  STRUCT
   FAC1_IF : STRUCT
    FAC_COMM_CHECK : INT ;	//FAC-PLC통신 확인용 정보 FAC=11,PLC=1
    PLC_ONLINE_MODE : INT ;	//생산지시 ON_OFF선택 정보 ON=1,OFF=0
    STATION_WORK_COMPLETE : INT ;	//공정 작업완료 정보 ON=1,OFF=0
    PLC_DATA_REQ_COUNT : INT ;	//차종 요청 카운터
    FINAL_SEND_VINDATA1 : WORD ;	//공정 최종 사용 VIN1
    FINAL_SEND_VINDATA2 : WORD ;	//공정 최종 사용 VIN2
    RCV_DATA_CHECK_ERROR : INT ;	//수신 데이터 CHECK이상 이상=1,정상=0
    RESERVED1 : INT ;
    RESERVED2 : INT ;
    RESERVED3 : INT ;
    LINE_DATA_READ_REQ : INT ;	//라인 현황 반영 요청 PLC=1,FAC=11
    ORDER_DATA_REQ : INT ;	//차종 설정 요청 PLC=1,FAC=11(정상처리),11<> 이상처리,99=서열부족,100=강제설정
    PRESENT_VIN_DATA1 : WORD ;	//차종 설정 데이터(현재)
    PRESENT_VIN_DATA2 : WORD ;	//차종 설정 데이터(현재)
    PRESENT_BODY_DATA1 : WORD ;	//차종 설정 데이터(현재)
    PRESENT_BODY_DATA2 : WORD ;	//차종 설정 데이터(현재)
    PRESENT_BODY_DATA3 : WORD ;	//차종 설정 데이터(현재)
    PRESENT_BODY_DATA4 : WORD ;	//차종 설정 데이터(현재)
    PRESENT_RESERVED_DATA1 : WORD ;	//차종 설정 데이터(현재)
    PRESENT_RESERVED_DATA2 : WORD ;	//차종 설정 데이터(현재)
    NEXT_VIN_DATA1 : WORD ;	//차종 설정 데이터(다음)
    NEXT_VIN_DATA2 : WORD ;	//차종 설정 데이터(다음)
    NEXT_BODY_DATA1 : WORD ;	//차종 설정 데이터(다음)
    NEXT_BODY_DATA2 : WORD ;	//차종 설정 데이터(다음)
    NEXT_BODY_DATA3 : WORD ;	//차종 설정 데이터(다음)
    NEXT_BODY_DATA4 : WORD ;	//차종 설정 데이터(다음)
    NEXT_RESERVED_DATA1 : WORD ;	//차종 설정 데이터(다음)
    NEXT_RESERVED_DATA2 : WORD ;	//차종 설정 데이터(다음)
    RESERVED4 : WORD ;
    RESERVED5 : WORD ;
   END_STRUCT ;
   FAC2_IF : STRUCT
    FAC_COMM_CHECK : INT ;	//FAC-PLC통신 확인용 정보 FAC=11,PLC=1
    PLC_ONLINE_MODE : INT ;	//생산지시 ON_OFF선택 정보 ON=1,OFF=0
    STATION_WORK_COMPLETE : INT ;	//공정 작업완료 정보 ON=1,OFF=0
    PLC_DATA_REQ_COUNT : INT ;	//차종 요청 카운터
    FINAL_SEND_VINDATA1 : WORD ;	//공정 최종 사용 VIN1
    FINAL_SEND_VINDATA2 : WORD ;	//공정 최종 사용 VIN2
    RCV_DATA_CHECK_ERROR : INT ;	//수신 데이터 CHECK이상 이상=1,정상=0
    RESERVED1 : INT ;
    RESERVED2 : INT ;
    CMP_ORDER_DATA_REQ : INT ;	//차종 설정 요청 정보 변경 내용 확인용
    LINE_DATA_READ_REQ : INT ;	//라인 현황 반영 요청 PLC=1,FAC=11
    ORDER_DATA_REQ : INT ;	//차종 설정 요청 PLC=1,FAC=11(정상처리),11<> 이상처리,99=서열부족,100=강제설정
    PRESENT_VIN_DATA1 : WORD ;	//차종 설정 데이터(현재)
    PRESENT_VIN_DATA2 : WORD ;	//차종 설정 데이터(현재)
    PRESENT_BODY_DATA1 : WORD ;	//차종 설정 데이터(현재)
    PRESENT_BODY_DATA : WORD ;	//차종 설정 데이터(현재)
    PRESENT_BODY_DATA3 : WORD ;	//차종 설정 데이터(현재)
    PRESENT_BODY_DATA4 : WORD ;	//차종 설정 데이터(현재)
    PRESENT_RESERVED_DATA1 : WORD ;	//차종 설정 데이터(현재)
    PRESENT_RESERVED_DATA2 : WORD ;	//차종 설정 데이터(현재)
    NEXT_VIN_DATA1 : WORD ;	//차종 설정 데이터(다음)
    NEXT_VIN_DATA2 : WORD ;	//차종 설정 데이터(다음)
    NEXT_BODY_DATA1 : WORD ;	//차종 설정 데이터(다음)
    NEXT_BODY_DATA2 : WORD ;	//차종 설정 데이터(다음)
    NEXT_BODY_DATA3 : WORD ;	//차종 설정 데이터(다음)
    NEXT_BODY_DATA4 : WORD ;	//차종 설정 데이터(다음)
    NEXT_RESERVED_DATA1 : WORD ;	//차종 설정 데이터(다음)
    NEXT_RESERVED_DATA2 : WORD ;	//차종 설정 데이터(다음)
    RESERVED4 : WORD ;
    RESERVED5 : WORD ;
   END_STRUCT ;
   FAC3_IF : STRUCT
    FAC_COMM_CHECK : INT ;	//FAC-PLC통신 확인용 정보 FAC=11,PLC=1
    PLC_ONLINE_MODE : INT ;	//생산지시 ON_OFF선택 정보 ON=1,OFF=0
    STATION_WORK_COMPLETE : INT ;	//공정 작업완료 정보 ON=1,OFF=0
    PLC_DATA_REQ_COUNT : INT ;	//차종 요청 카운터
    FINAL_SEND_VINDATA1 : WORD ;	//공정 최종 사용 VIN1
    FINAL_SEND_VINDATA2 : WORD ;	//공정 최종 사용 VIN2
    RCV_DATA_CHECK_ERROR : INT ;	//수신 데이터 CHECK이상 이상=1,정상=0
    RESERVED1 : INT ;
    RESERVED2 : INT ;
    CMP_ORDER_DATA_REQ : INT ;	//차종 설정 요청 정보 변경 내용 확인용
    LINE_DATA_READ_REQ : INT ;	//라인 현황 반영 요청 PLC=1,FAC=11
    ORDER_DATA_REQ : INT ;	//차종 설정 요청 PLC=1,FAC=11(정상처리),11<> 이상처리,99=서열부족,100=강제설정
    PRESENT_VIN_DATA1 : WORD ;	//차종 설정 데이터(현재)
    PRESENT_VIN_DATA2 : WORD ;	//차종 설정 데이터(현재)
    PRESENT_BODY_DATA1 : WORD ;	//차종 설정 데이터(현재)
    PRESENT_BODY_DATA : WORD ;	//차종 설정 데이터(현재)
    PRESENT_BODY_DATA3 : WORD ;	//차종 설정 데이터(현재)
    PRESENT_BODY_DATA4 : WORD ;	//차종 설정 데이터(현재)
    PRESENT_RESERVED_DATA1 : WORD ;	//차종 설정 데이터(현재)
    PRESENT_RESERVED_DATA2 : WORD ;	//차종 설정 데이터(현재)
    NEXT_VIN_DATA1 : WORD ;	//차종 설정 데이터(다음)
    NEXT_VIN_DATA2 : WORD ;	//차종 설정 데이터(다음)
    NEXT_BODY_DATA1 : WORD ;	//차종 설정 데이터(다음)
    NEXT_BODY_DATA2 : WORD ;	//차종 설정 데이터(다음)
    NEXT_BODY_DATA3 : WORD ;	//차종 설정 데이터(다음)
    NEXT_BODY_DATA4 : WORD ;	//차종 설정 데이터(다음)
    NEXT_RESERVED_DATA1 : WORD ;	//차종 설정 데이터(다음)
    NEXT_RESERVED_DATA2 : WORD ;	//차종 설정 데이터(다음)
    RESERVED4 : WORD ;
    RESERVED5 : WORD ;
   END_STRUCT ;
   FAC4_IF : STRUCT
    FAC_COMM_CHECK : INT ;	//FAC-PLC통신 확인용 정보 FAC=11,PLC=1
    PLC_ONLINE_MODE : INT ;	//생산지시 ON_OFF선택 정보 ON=1,OFF=0
    STATION_WORK_COMPLETE : INT ;	//공정 작업완료 정보 ON=1,OFF=0
    PLC_DATA_REQ_COUNT : INT ;	//차종 요청 카운터
    FINAL_SEND_VINDATA1 : WORD ;	//공정 최종 사용 VIN1
    FINAL_SEND_VINDATA2 : WORD ;	//공정 최종 사용 VIN2
    RCV_DATA_CHECK_ERROR : INT ;	//수신 데이터 CHECK이상 이상=1,정상=0
    RESERVED1 : INT ;
    RESERVED2 : INT ;
    CMP_ORDER_DATA_REQ : INT ;	//차종 설정 요청 정보 변경 내용 확인용
    LINE_DATA_READ_REQ : INT ;	//라인 현황 반영 요청 PLC=1,FAC=11
    ORDER_DATA_REQ : INT ;	//차종 설정 요청 PLC=1,FAC=11(정상처리),11<> 이상처리,99=서열부족,100=강제설정
    PRESENT_VIN_DATA1 : WORD ;	//차종 설정 데이터(현재)
    PRESENT_VIN_DATA2 : WORD ;	//차종 설정 데이터(현재)
    PRESENT_BODY_DATA1 : WORD ;	//차종 설정 데이터(현재)
    PRESENT_BODY_DATA : WORD ;	//차종 설정 데이터(현재)
    PRESENT_BODY_DATA3 : WORD ;	//차종 설정 데이터(현재)
    PRESENT_BODY_DATA4 : WORD ;	//차종 설정 데이터(현재)
    PRESENT_RESERVED_DATA1 : WORD ;	//차종 설정 데이터(현재)
    PRESENT_RESERVED_DATA2 : WORD ;	//차종 설정 데이터(현재)
    NEXT_VIN_DATA1 : WORD ;	//차종 설정 데이터(다음)
    NEXT_VIN_DATA2 : WORD ;	//차종 설정 데이터(다음)
    NEXT_BODY_DATA1 : WORD ;	//차종 설정 데이터(다음)
    NEXT_BODY_DATA2 : WORD ;	//차종 설정 데이터(다음)
    NEXT_BODY_DATA3 : WORD ;	//차종 설정 데이터(다음)
    NEXT_BODY_DATA4 : WORD ;	//차종 설정 데이터(다음)
    NEXT_RESERVED_DATA1 : WORD ;	//차종 설정 데이터(다음)
    NEXT_RESERVED_DATA2 : WORD ;	//차종 설정 데이터(다음)
    RESERVED4 : WORD ;
    RESERVED5 : WORD ;
   END_STRUCT ;
   FAC5_IF : STRUCT
    FAC_COMM_CHECK : INT ;	//FAC-PLC통신 확인용 정보 FAC=11,PLC=1
    PLC_ONLINE_MODE : INT ;	//생산지시 ON_OFF선택 정보 ON=1,OFF=0
    STATION_WORK_COMPLETE : INT ;	//공정 작업완료 정보 ON=1,OFF=0
    PLC_DATA_REQ_COUNT : INT ;	//차종 요청 카운터
    FINAL_SEND_VINDATA1 : WORD ;	//공정 최종 사용 VIN1
    FINAL_SEND_VINDATA2 : WORD ;	//공정 최종 사용 VIN2
    RCV_DATA_CHECK_ERROR : INT ;	//수신 데이터 CHECK이상 이상=1,정상=0
    RESERVED1 : INT ;
    RESERVED2 : INT ;
    CMP_ORDER_DATA_REQ : INT ;	//차종 설정 요청 정보 변경 내용 확인용
    LINE_DATA_READ_REQ : INT ;	//라인 현황 반영 요청 PLC=1,FAC=11
    ORDER_DATA_REQ : INT ;	//차종 설정 요청 PLC=1,FAC=11(정상처리),11<> 이상처리,99=서열부족,100=강제설정
    PRESENT_VIN_DATA1 : WORD ;	//차종 설정 데이터(현재)
    PRESENT_VIN_DATA2 : WORD ;	//차종 설정 데이터(현재)
    PRESENT_BODY_DATA1 : WORD ;	//차종 설정 데이터(현재)
    PRESENT_BODY_DATA : WORD ;	//차종 설정 데이터(현재)
    PRESENT_BODY_DATA3 : WORD ;	//차종 설정 데이터(현재)
    PRESENT_BODY_DATA4 : WORD ;	//차종 설정 데이터(현재)
    PRESENT_RESERVED_DATA1 : WORD ;	//차종 설정 데이터(현재)
    PRESENT_RESERVED_DATA2 : WORD ;	//차종 설정 데이터(현재)
    NEXT_VIN_DATA1 : WORD ;	//차종 설정 데이터(다음)
    NEXT_VIN_DATA2 : WORD ;	//차종 설정 데이터(다음)
    NEXT_BODY_DATA1 : WORD ;	//차종 설정 데이터(다음)
    NEXT_BODY_DATA2 : WORD ;	//차종 설정 데이터(다음)
    NEXT_BODY_DATA3 : WORD ;	//차종 설정 데이터(다음)
    NEXT_BODY_DATA4 : WORD ;	//차종 설정 데이터(다음)
    NEXT_RESERVED_DATA1 : WORD ;	//차종 설정 데이터(다음)
    NEXT_RESERVED_DATA2 : WORD ;	//차종 설정 데이터(다음)
    RESERVED4 : WORD ;
    RESERVED5 : WORD ;
   END_STRUCT ;
   FAC6_IF : STRUCT
    FAC_COMM_CHECK : INT ;	//FAC-PLC통신 확인용 정보 FAC=11,PLC=1
    PLC_ONLINE_MODE : INT ;	//생산지시 ON_OFF선택 정보 ON=1,OFF=0
    STATION_WORK_COMPLETE : INT ;	//공정 작업완료 정보 ON=1,OFF=0
    PLC_DATA_REQ_COUNT : INT ;	//차종 요청 카운터
    FINAL_SEND_VINDATA1 : WORD ;	//공정 최종 사용 VIN1
    FINAL_SEND_VINDATA2 : WORD ;	//공정 최종 사용 VIN2
    RCV_DATA_CHECK_ERROR : INT ;	//수신 데이터 CHECK이상 이상=1,정상=0
    RESERVED1 : INT ;
    RESERVED2 : INT ;
    CMP_ORDER_DATA_REQ : INT ;	//차종 설정 요청 정보 변경 내용 확인용
    LINE_DATA_READ_REQ : INT ;	//라인 현황 반영 요청 PLC=1,FAC=11
    ORDER_DATA_REQ : INT ;	//차종 설정 요청 PLC=1,FAC=11(정상처리),11<> 이상처리,99=서열부족,100=강제설정
    PRESENT_VIN_DATA1 : WORD ;	//차종 설정 데이터(현재)
    PRESENT_VIN_DATA2 : WORD ;	//차종 설정 데이터(현재)
    PRESENT_BODY_DATA1 : WORD ;	//차종 설정 데이터(현재)
    PRESENT_BODY_DATA : WORD ;	//차종 설정 데이터(현재)
    PRESENT_BODY_DATA3 : WORD ;	//차종 설정 데이터(현재)
    PRESENT_BODY_DATA4 : WORD ;	//차종 설정 데이터(현재)
    PRESENT_RESERVED_DATA1 : WORD ;	//차종 설정 데이터(현재)
    PRESENT_RESERVED_DATA2 : WORD ;	//차종 설정 데이터(현재)
    NEXT_VIN_DATA1 : WORD ;	//차종 설정 데이터(다음)
    NEXT_VIN_DATA2 : WORD ;	//차종 설정 데이터(다음)
    NEXT_BODY_DATA1 : WORD ;	//차종 설정 데이터(다음)
    NEXT_BODY_DATA2 : WORD ;	//차종 설정 데이터(다음)
    NEXT_BODY_DATA3 : WORD ;	//차종 설정 데이터(다음)
    NEXT_BODY_DATA4 : WORD ;	//차종 설정 데이터(다음)
    NEXT_RESERVED_DATA1 : WORD ;	//차종 설정 데이터(다음)
    NEXT_RESERVED_DATA2 : WORD ;	//차종 설정 데이터(다음)
    RESERVED4 : WORD ;
    RESERVED5 : WORD ;
   END_STRUCT ;
   FAC7_IF : STRUCT
    FAC_COMM_CHECK : INT ;	//FAC-PLC통신 확인용 정보 FAC=11,PLC=1
    PLC_ONLINE_MODE : INT ;	//생산지시 ON_OFF선택 정보 ON=1,OFF=0
    STATION_WORK_COMPLETE : INT ;	//공정 작업완료 정보 ON=1,OFF=0
    PLC_DATA_REQ_COUNT : INT ;	//차종 요청 카운터
    FINAL_SEND_VINDATA1 : WORD ;	//공정 최종 사용 VIN1
    FINAL_SEND_VINDATA2 : WORD ;	//공정 최종 사용 VIN2
    RCV_DATA_CHECK_ERROR : INT ;	//수신 데이터 CHECK이상 이상=1,정상=0
    RESERVED1 : INT ;
    RESERVED2 : INT ;
    CMP_ORDER_DATA_REQ : INT ;	//차종 설정 요청 정보 변경 내용 확인용
    LINE_DATA_READ_REQ : INT ;	//라인 현황 반영 요청 PLC=1,FAC=11
    ORDER_DATA_REQ : INT ;	//차종 설정 요청 PLC=1,FAC=11(정상처리),11<> 이상처리,99=서열부족,100=강제설정
    PRESENT_VIN_DATA1 : WORD ;	//차종 설정 데이터(현재)
    PRESENT_VIN_DATA2 : WORD ;	//차종 설정 데이터(현재)
    PRESENT_BODY_DATA1 : WORD ;	//차종 설정 데이터(현재)
    PRESENT_BODY_DATA : WORD ;	//차종 설정 데이터(현재)
    PRESENT_BODY_DATA3 : WORD ;	//차종 설정 데이터(현재)
    PRESENT_BODY_DATA4 : WORD ;	//차종 설정 데이터(현재)
    PRESENT_RESERVED_DATA1 : WORD ;	//차종 설정 데이터(현재)
    PRESENT_RESERVED_DATA2 : WORD ;	//차종 설정 데이터(현재)
    NEXT_VIN_DATA1 : WORD ;	//차종 설정 데이터(다음)
    NEXT_VIN_DATA2 : WORD ;	//차종 설정 데이터(다음)
    NEXT_BODY_DATA1 : WORD ;	//차종 설정 데이터(다음)
    NEXT_BODY_DATA2 : WORD ;	//차종 설정 데이터(다음)
    NEXT_BODY_DATA3 : WORD ;	//차종 설정 데이터(다음)
    NEXT_BODY_DATA4 : WORD ;	//차종 설정 데이터(다음)
    NEXT_RESERVED_DATA1 : WORD ;	//차종 설정 데이터(다음)
    NEXT_RESERVED_DATA2 : WORD ;	//차종 설정 데이터(다음)
    RESERVED4 : WORD ;
    RESERVED5 : WORD ;
   END_STRUCT ;
   FAC8_IF : STRUCT
    FAC_COMM_CHECK : INT ;	//FAC-PLC통신 확인용 정보 FAC=11,PLC=1
    PLC_ONLINE_MODE : INT ;	//생산지시 ON_OFF선택 정보 ON=1,OFF=0
    STATION_WORK_COMPLETE : INT ;	//공정 작업완료 정보 ON=1,OFF=0
    PLC_DATA_REQ_COUNT : INT ;	//차종 요청 카운터
    FINAL_SEND_VINDATA1 : WORD ;	//공정 최종 사용 VIN1
    FINAL_SEND_VINDATA2 : WORD ;	//공정 최종 사용 VIN2
    RCV_DATA_CHECK_ERROR : INT ;	//수신 데이터 CHECK이상 이상=1,정상=0
    RESERVED1 : INT ;
    RESERVED2 : INT ;
    CMP_ORDER_DATA_REQ : INT ;	//차종 설정 요청 정보 변경 내용 확인용
    LINE_DATA_READ_REQ : INT ;	//라인 현황 반영 요청 PLC=1,FAC=11
    ORDER_DATA_REQ : INT ;	//차종 설정 요청 PLC=1,FAC=11(정상처리),11<> 이상처리,99=서열부족,100=강제설정
    PRESENT_VIN_DATA1 : WORD ;	//차종 설정 데이터(현재)
    PRESENT_VIN_DATA2 : WORD ;	//차종 설정 데이터(현재)
    PRESENT_BODY_DATA1 : WORD ;	//차종 설정 데이터(현재)
    PRESENT_BODY_DATA : WORD ;	//차종 설정 데이터(현재)
    PRESENT_BODY_DATA3 : WORD ;	//차종 설정 데이터(현재)
    PRESENT_BODY_DATA4 : WORD ;	//차종 설정 데이터(현재)
    PRESENT_RESERVED_DATA1 : WORD ;	//차종 설정 데이터(현재)
    PRESENT_RESERVED_DATA2 : WORD ;	//차종 설정 데이터(현재)
    NEXT_VIN_DATA1 : WORD ;	//차종 설정 데이터(다음)
    NEXT_VIN_DATA2 : WORD ;	//차종 설정 데이터(다음)
    NEXT_BODY_DATA1 : WORD ;	//차종 설정 데이터(다음)
    NEXT_BODY_DATA2 : WORD ;	//차종 설정 데이터(다음)
    NEXT_BODY_DATA3 : WORD ;	//차종 설정 데이터(다음)
    NEXT_BODY_DATA4 : WORD ;	//차종 설정 데이터(다음)
    NEXT_RESERVED_DATA1 : WORD ;	//차종 설정 데이터(다음)
    NEXT_RESERVED_DATA2 : WORD ;	//차종 설정 데이터(다음)
    RESERVED4 : WORD ;
    RESERVED5 : WORD ;
   END_STRUCT ;
   FAC9_IF : STRUCT
    FAC_COMM_CHECK : INT ;	//FAC-PLC통신 확인용 정보 FAC=11,PLC=1
    PLC_ONLINE_MODE : INT ;	//생산지시 ON_OFF선택 정보 ON=1,OFF=0
    STATION_WORK_COMPLETE : INT ;	//공정 작업완료 정보 ON=1,OFF=0
    PLC_DATA_REQ_COUNT : INT ;	//차종 요청 카운터
    FINAL_SEND_VINDATA1 : WORD ;	//공정 최종 사용 VIN1
    FINAL_SEND_VINDATA2 : WORD ;	//공정 최종 사용 VIN2
    RCV_DATA_CHECK_ERROR : INT ;	//수신 데이터 CHECK이상 이상=1,정상=0
    RESERVED1 : INT ;
    RESERVED2 : INT ;
    CMP_ORDER_DATA_REQ : INT ;	//차종 설정 요청 정보 변경 내용 확인용
    LINE_DATA_READ_REQ : INT ;	//라인 현황 반영 요청 PLC=1,FAC=11
    ORDER_DATA_REQ : INT ;	//차종 설정 요청 PLC=1,FAC=11(정상처리),11<> 이상처리,99=서열부족,100=강제설정
    PRESENT_VIN_DATA1 : WORD ;	//차종 설정 데이터(현재)
    PRESENT_VIN_DATA2 : WORD ;	//차종 설정 데이터(현재)
    PRESENT_BODY_DATA1 : WORD ;	//차종 설정 데이터(현재)
    PRESENT_BODY_DATA : WORD ;	//차종 설정 데이터(현재)
    PRESENT_BODY_DATA3 : WORD ;	//차종 설정 데이터(현재)
    PRESENT_BODY_DATA4 : WORD ;	//차종 설정 데이터(현재)
    PRESENT_RESERVED_DATA1 : WORD ;	//차종 설정 데이터(현재)
    PRESENT_RESERVED_DATA2 : WORD ;	//차종 설정 데이터(현재)
    NEXT_VIN_DATA1 : WORD ;	//차종 설정 데이터(다음)
    NEXT_VIN_DATA2 : WORD ;	//차종 설정 데이터(다음)
    NEXT_BODY_DATA1 : WORD ;	//차종 설정 데이터(다음)
    NEXT_BODY_DATA2 : WORD ;	//차종 설정 데이터(다음)
    NEXT_BODY_DATA3 : WORD ;	//차종 설정 데이터(다음)
    NEXT_BODY_DATA4 : WORD ;	//차종 설정 데이터(다음)
    NEXT_RESERVED_DATA1 : WORD ;	//차종 설정 데이터(다음)
    NEXT_RESERVED_DATA2 : WORD ;	//차종 설정 데이터(다음)
    RESERVED4 : WORD ;
    RESERVED5 : WORD ;
   END_STRUCT ;
   FAC10_IF : STRUCT
    FAC_COMM_CHECK : INT ;	//FAC-PLC통신 확인용 정보 FAC=11,PLC=1
    PLC_ONLINE_MODE : INT ;	//생산지시 ON_OFF선택 정보 ON=1,OFF=0
    STATION_WORK_COMPLETE : INT ;	//공정 작업완료 정보 ON=1,OFF=0
    PLC_DATA_REQ_COUNT : INT ;	//차종 요청 카운터
    FINAL_SEND_VINDATA1 : WORD ;	//공정 최종 사용 VIN1
    FINAL_SEND_VINDATA2 : WORD ;	//공정 최종 사용 VIN2
    RCV_DATA_CHECK_ERROR : INT ;	//수신 데이터 CHECK이상 이상=1,정상=0
    RESERVED1 : INT ;
    RESERVED2 : INT ;
    CMP_ORDER_DATA_REQ : INT ;	//차종 설정 요청 정보 변경 내용 확인용
    LINE_DATA_READ_REQ : INT ;	//라인 현황 반영 요청 PLC=1,FAC=11
    ORDER_DATA_REQ : INT ;	//차종 설정 요청 PLC=1,FAC=11(정상처리),11<> 이상처리,99=서열부족,100=강제설정
    PRESENT_VIN_DATA1 : WORD ;	//차종 설정 데이터(현재)
    PRESENT_VIN_DATA2 : WORD ;	//차종 설정 데이터(현재)
    PRESENT_BODY_DATA1 : WORD ;	//차종 설정 데이터(현재)
    PRESENT_BODY_DATA : WORD ;	//차종 설정 데이터(현재)
    PRESENT_BODY_DATA3 : WORD ;	//차종 설정 데이터(현재)
    PRESENT_BODY_DATA4 : WORD ;	//차종 설정 데이터(현재)
    PRESENT_RESERVED_DATA1 : WORD ;	//차종 설정 데이터(현재)
    PRESENT_RESERVED_DATA2 : WORD ;	//차종 설정 데이터(현재)
    NEXT_VIN_DATA1 : WORD ;	//차종 설정 데이터(다음)
    NEXT_VIN_DATA2 : WORD ;	//차종 설정 데이터(다음)
    NEXT_BODY_DATA1 : WORD ;	//차종 설정 데이터(다음)
    NEXT_BODY_DATA2 : WORD ;	//차종 설정 데이터(다음)
    NEXT_BODY_DATA3 : WORD ;	//차종 설정 데이터(다음)
    NEXT_BODY_DATA4 : WORD ;	//차종 설정 데이터(다음)
    NEXT_RESERVED_DATA1 : WORD ;	//차종 설정 데이터(다음)
    NEXT_RESERVED_DATA2 : WORD ;	//차종 설정 데이터(다음)
    RESERVED4 : WORD ;
    RESERVED5 : WORD ;
   END_STRUCT ;
   FAC11_IF : STRUCT
    FAC_COMM_CHECK : INT ;	//FAC-PLC통신 확인용 정보 FAC=11,PLC=1
    PLC_ONLINE_MODE : INT ;	//생산지시 ON_OFF선택 정보 ON=1,OFF=0
    STATION_WORK_COMPLETE : INT ;	//공정 작업완료 정보 ON=1,OFF=0
    PLC_DATA_REQ_COUNT : INT ;	//차종 요청 카운터
    FINAL_SEND_VINDATA1 : WORD ;	//공정 최종 사용 VIN1
    FINAL_SEND_VINDATA2 : WORD ;	//공정 최종 사용 VIN2
    RCV_DATA_CHECK_ERROR : INT ;	//수신 데이터 CHECK이상 이상=1,정상=0
    RESERVED1 : INT ;
    RESERVED2 : INT ;
    CMP_ORDER_DATA_REQ : INT ;	//차종 설정 요청 정보 변경 내용 확인용
    LINE_DATA_READ_REQ : INT ;	//라인 현황 반영 요청 PLC=1,FAC=11
    ORDER_DATA_REQ : INT ;	//차종 설정 요청 PLC=1,FAC=11(정상처리),11<> 이상처리,99=서열부족,100=강제설정
    PRESENT_VIN_DATA1 : WORD ;	//차종 설정 데이터(현재)
    PRESENT_VIN_DATA2 : WORD ;	//차종 설정 데이터(현재)
    PRESENT_BODY_DATA1 : WORD ;	//차종 설정 데이터(현재)
    PRESENT_BODY_DATA : WORD ;	//차종 설정 데이터(현재)
    PRESENT_BODY_DATA3 : WORD ;	//차종 설정 데이터(현재)
    PRESENT_BODY_DATA4 : WORD ;	//차종 설정 데이터(현재)
    PRESENT_RESERVED_DATA1 : WORD ;	//차종 설정 데이터(현재)
    PRESENT_RESERVED_DATA2 : WORD ;	//차종 설정 데이터(현재)
    NEXT_VIN_DATA1 : WORD ;	//차종 설정 데이터(다음)
    NEXT_VIN_DATA2 : WORD ;	//차종 설정 데이터(다음)
    NEXT_BODY_DATA1 : WORD ;	//차종 설정 데이터(다음)
    NEXT_BODY_DATA2 : WORD ;	//차종 설정 데이터(다음)
    NEXT_BODY_DATA3 : WORD ;	//차종 설정 데이터(다음)
    NEXT_BODY_DATA4 : WORD ;	//차종 설정 데이터(다음)
    NEXT_RESERVED_DATA1 : WORD ;	//차종 설정 데이터(다음)
    NEXT_RESERVED_DATA2 : WORD ;	//차종 설정 데이터(다음)
    RESERVED4 : WORD ;
    RESERVED5 : WORD ;
   END_STRUCT ;
   FAC12_IF : STRUCT
    FAC_COMM_CHECK : INT ;	//FAC-PLC통신 확인용 정보 FAC=11,PLC=1
    PLC_ONLINE_MODE : INT ;	//생산지시 ON_OFF선택 정보 ON=1,OFF=0
    STATION_WORK_COMPLETE : INT ;	//공정 작업완료 정보 ON=1,OFF=0
    PLC_DATA_REQ_COUNT : INT ;	//차종 요청 카운터
    FINAL_SEND_VINDATA1 : WORD ;	//공정 최종 사용 VIN1
    FINAL_SEND_VINDATA2 : WORD ;	//공정 최종 사용 VIN2
    RCV_DATA_CHECK_ERROR : INT ;	//수신 데이터 CHECK이상 이상=1,정상=0
    RESERVED1 : INT ;
    RESERVED2 : INT ;
    CMP_ORDER_DATA_REQ : INT ;	//차종 설정 요청 정보 변경 내용 확인용
    LINE_DATA_READ_REQ : INT ;	//라인 현황 반영 요청 PLC=1,FAC=11
    ORDER_DATA_REQ : INT ;	//차종 설정 요청 PLC=1,FAC=11(정상처리),11<> 이상처리,99=서열부족,100=강제설정
    PRESENT_VIN_DATA1 : WORD ;	//차종 설정 데이터(현재)
    PRESENT_VIN_DATA2 : WORD ;	//차종 설정 데이터(현재)
    PRESENT_BODY_DATA1 : WORD ;	//차종 설정 데이터(현재)
    PRESENT_BODY_DATA : WORD ;	//차종 설정 데이터(현재)
    PRESENT_BODY_DATA3 : WORD ;	//차종 설정 데이터(현재)
    PRESENT_BODY_DATA4 : WORD ;	//차종 설정 데이터(현재)
    PRESENT_RESERVED_DATA1 : WORD ;	//차종 설정 데이터(현재)
    PRESENT_RESERVED_DATA2 : WORD ;	//차종 설정 데이터(현재)
    NEXT_VIN_DATA1 : WORD ;	//차종 설정 데이터(다음)
    NEXT_VIN_DATA2 : WORD ;	//차종 설정 데이터(다음)
    NEXT_BODY_DATA1 : WORD ;	//차종 설정 데이터(다음)
    NEXT_BODY_DATA2 : WORD ;	//차종 설정 데이터(다음)
    NEXT_BODY_DATA3 : WORD ;	//차종 설정 데이터(다음)
    NEXT_BODY_DATA4 : WORD ;	//차종 설정 데이터(다음)
    NEXT_RESERVED_DATA1 : WORD ;	//차종 설정 데이터(다음)
    NEXT_RESERVED_DATA2 : WORD ;	//차종 설정 데이터(다음)
    RESERVED4 : WORD ;
    RESERVED5 : WORD ;
   END_STRUCT ;
   FAC13_IF : STRUCT
    FAC_COMM_CHECK : INT ;	//FAC-PLC통신 확인용 정보 FAC=11,PLC=1
    PLC_ONLINE_MODE : INT ;	//생산지시 ON_OFF선택 정보 ON=1,OFF=0
    STATION_WORK_COMPLETE : INT ;	//공정 작업완료 정보 ON=1,OFF=0
    PLC_DATA_REQ_COUNT : INT ;	//차종 요청 카운터
    FINAL_SEND_VINDATA1 : WORD ;	//공정 최종 사용 VIN1
    FINAL_SEND_VINDATA2 : WORD ;	//공정 최종 사용 VIN2
    RCV_DATA_CHECK_ERROR : INT ;	//수신 데이터 CHECK이상 이상=1,정상=0
    RESERVED1 : INT ;
    RESERVED2 : INT ;
    CMP_ORDER_DATA_REQ : INT ;	//차종 설정 요청 정보 변경 내용 확인용
    LINE_DATA_READ_REQ : INT ;	//라인 현황 반영 요청 PLC=1,FAC=11
    ORDER_DATA_REQ : INT ;	//차종 설정 요청 PLC=1,FAC=11(정상처리),11<> 이상처리,99=서열부족,100=강제설정
    PRESENT_VIN_DATA1 : WORD ;	//차종 설정 데이터(현재)
    PRESENT_VIN_DATA2 : WORD ;	//차종 설정 데이터(현재)
    PRESENT_BODY_DATA1 : WORD ;	//차종 설정 데이터(현재)
    PRESENT_BODY_DATA : WORD ;	//차종 설정 데이터(현재)
    PRESENT_BODY_DATA3 : WORD ;	//차종 설정 데이터(현재)
    PRESENT_BODY_DATA4 : WORD ;	//차종 설정 데이터(현재)
    PRESENT_RESERVED_DATA1 : WORD ;	//차종 설정 데이터(현재)
    PRESENT_RESERVED_DATA2 : WORD ;	//차종 설정 데이터(현재)
    NEXT_VIN_DATA1 : WORD ;	//차종 설정 데이터(다음)
    NEXT_VIN_DATA2 : WORD ;	//차종 설정 데이터(다음)
    NEXT_BODY_DATA1 : WORD ;	//차종 설정 데이터(다음)
    NEXT_BODY_DATA2 : WORD ;	//차종 설정 데이터(다음)
    NEXT_BODY_DATA3 : WORD ;	//차종 설정 데이터(다음)
    NEXT_BODY_DATA4 : WORD ;	//차종 설정 데이터(다음)
    NEXT_RESERVED_DATA1 : WORD ;	//차종 설정 데이터(다음)
    NEXT_RESERVED_DATA2 : WORD ;	//차종 설정 데이터(다음)
    RESERVED4 : WORD ;
    RESERVED5 : WORD ;
   END_STRUCT ;
   FAC14_IF : STRUCT
    FAC_COMM_CHECK : INT ;	//FAC-PLC통신 확인용 정보 FAC=11,PLC=1
    PLC_ONLINE_MODE : INT ;	//생산지시 ON_OFF선택 정보 ON=1,OFF=0
    STATION_WORK_COMPLETE : INT ;	//공정 작업완료 정보 ON=1,OFF=0
    PLC_DATA_REQ_COUNT : INT ;	//차종 요청 카운터
    FINAL_SEND_VINDATA1 : WORD ;	//공정 최종 사용 VIN1
    FINAL_SEND_VINDATA2 : WORD ;	//공정 최종 사용 VIN2
    RCV_DATA_CHECK_ERROR : INT ;	//수신 데이터 CHECK이상 이상=1,정상=0
    RESERVED1 : INT ;
    RESERVED2 : INT ;
    CMP_ORDER_DATA_REQ : INT ;	//차종 설정 요청 정보 변경 내용 확인용
    LINE_DATA_READ_REQ : INT ;	//라인 현황 반영 요청 PLC=1,FAC=11
    ORDER_DATA_REQ : INT ;	//차종 설정 요청 PLC=1,FAC=11(정상처리),11<> 이상처리,99=서열부족,100=강제설정
    PRESENT_VIN_DATA1 : WORD ;	//차종 설정 데이터(현재)
    PRESENT_VIN_DATA2 : WORD ;	//차종 설정 데이터(현재)
    PRESENT_BODY_DATA1 : WORD ;	//차종 설정 데이터(현재)
    PRESENT_BODY_DATA : WORD ;	//차종 설정 데이터(현재)
    PRESENT_BODY_DATA3 : WORD ;	//차종 설정 데이터(현재)
    PRESENT_BODY_DATA4 : WORD ;	//차종 설정 데이터(현재)
    PRESENT_RESERVED_DATA1 : WORD ;	//차종 설정 데이터(현재)
    PRESENT_RESERVED_DATA2 : WORD ;	//차종 설정 데이터(현재)
    NEXT_VIN_DATA1 : WORD ;	//차종 설정 데이터(다음)
    NEXT_VIN_DATA2 : WORD ;	//차종 설정 데이터(다음)
    NEXT_BODY_DATA1 : WORD ;	//차종 설정 데이터(다음)
    NEXT_BODY_DATA2 : WORD ;	//차종 설정 데이터(다음)
    NEXT_BODY_DATA3 : WORD ;	//차종 설정 데이터(다음)
    NEXT_BODY_DATA4 : WORD ;	//차종 설정 데이터(다음)
    NEXT_RESERVED_DATA1 : WORD ;	//차종 설정 데이터(다음)
    NEXT_RESERVED_DATA2 : WORD ;	//차종 설정 데이터(다음)
    RESERVED4 : WORD ;
    RESERVED5 : WORD ;
   END_STRUCT ;
   FAC15_IF : STRUCT
    FAC_COMM_CHECK : INT ;	//FAC-PLC통신 확인용 정보 FAC=11,PLC=1
    PLC_ONLINE_MODE : INT ;	//생산지시 ON_OFF선택 정보 ON=1,OFF=0
    STATION_WORK_COMPLETE : INT ;	//공정 작업완료 정보 ON=1,OFF=0
    PLC_DATA_REQ_COUNT : INT ;	//차종 요청 카운터
    FINAL_SEND_VINDATA1 : WORD ;	//공정 최종 사용 VIN1
    FINAL_SEND_VINDATA2 : WORD ;	//공정 최종 사용 VIN2
    RCV_DATA_CHECK_ERROR : INT ;	//수신 데이터 CHECK이상 이상=1,정상=0
    RESERVED1 : INT ;
    RESERVED2 : INT ;
    CMP_ORDER_DATA_REQ : INT ;	//차종 설정 요청 정보 변경 내용 확인용
    LINE_DATA_READ_REQ : INT ;	//라인 현황 반영 요청 PLC=1,FAC=11
    ORDER_DATA_REQ : INT ;	//차종 설정 요청 PLC=1,FAC=11(정상처리),11<> 이상처리,99=서열부족,100=강제설정
    PRESENT_VIN_DATA1 : WORD ;	//차종 설정 데이터(현재)
    PRESENT_VIN_DATA2 : WORD ;	//차종 설정 데이터(현재)
    PRESENT_BODY_DATA1 : WORD ;	//차종 설정 데이터(현재)
    PRESENT_BODY_DATA : WORD ;	//차종 설정 데이터(현재)
    PRESENT_BODY_DATA3 : WORD ;	//차종 설정 데이터(현재)
    PRESENT_BODY_DATA4 : WORD ;	//차종 설정 데이터(현재)
    PRESENT_RESERVED_DATA1 : WORD ;	//차종 설정 데이터(현재)
    PRESENT_RESERVED_DATA2 : WORD ;	//차종 설정 데이터(현재)
    NEXT_VIN_DATA1 : WORD ;	//차종 설정 데이터(다음)
    NEXT_VIN_DATA2 : WORD ;	//차종 설정 데이터(다음)
    NEXT_BODY_DATA1 : WORD ;	//차종 설정 데이터(다음)
    NEXT_BODY_DATA2 : WORD ;	//차종 설정 데이터(다음)
    NEXT_BODY_DATA3 : WORD ;	//차종 설정 데이터(다음)
    NEXT_BODY_DATA4 : WORD ;	//차종 설정 데이터(다음)
    NEXT_RESERVED_DATA1 : WORD ;	//차종 설정 데이터(다음)
    NEXT_RESERVED_DATA2 : WORD ;	//차종 설정 데이터(다음)
    RESERVED4 : WORD ;
    RESERVED5 : WORD ;
   END_STRUCT ;
   FAC16_IF : STRUCT
    FAC_COMM_CHECK : INT ;	//FAC-PLC통신 확인용 정보 FAC=11,PLC=1
    PLC_ONLINE_MODE : INT ;	//생산지시 ON_OFF선택 정보 ON=1,OFF=0
    STATION_WORK_COMPLETE : INT ;	//공정 작업완료 정보 ON=1,OFF=0
    PLC_DATA_REQ_COUNT : INT ;	//차종 요청 카운터
    FINAL_SEND_VINDATA1 : WORD ;	//공정 최종 사용 VIN1
    FINAL_SEND_VINDATA2 : WORD ;	//공정 최종 사용 VIN2
    RCV_DATA_CHECK_ERROR : INT ;	//수신 데이터 CHECK이상 이상=1,정상=0
    RESERVED1 : INT ;
    RESERVED2 : INT ;
    CMP_ORDER_DATA_REQ : INT ;	//차종 설정 요청 정보 변경 내용 확인용
    LINE_DATA_READ_REQ : INT ;	//라인 현황 반영 요청 PLC=1,FAC=11
    ORDER_DATA_REQ : INT ;	//차종 설정 요청 PLC=1,FAC=11(정상처리),11<> 이상처리,99=서열부족,100=강제설정
    PRESENT_VIN_DATA1 : WORD ;	//차종 설정 데이터(현재)
    PRESENT_VIN_DATA2 : WORD ;	//차종 설정 데이터(현재)
    PRESENT_BODY_DATA1 : WORD ;	//차종 설정 데이터(현재)
    PRESENT_BODY_DATA : WORD ;	//차종 설정 데이터(현재)
    PRESENT_BODY_DATA3 : WORD ;	//차종 설정 데이터(현재)
    PRESENT_BODY_DATA4 : WORD ;	//차종 설정 데이터(현재)
    PRESENT_RESERVED_DATA1 : WORD ;	//차종 설정 데이터(현재)
    PRESENT_RESERVED_DATA2 : WORD ;	//차종 설정 데이터(현재)
    NEXT_VIN_DATA1 : WORD ;	//차종 설정 데이터(다음)
    NEXT_VIN_DATA2 : WORD ;	//차종 설정 데이터(다음)
    NEXT_BODY_DATA1 : WORD ;	//차종 설정 데이터(다음)
    NEXT_BODY_DATA2 : WORD ;	//차종 설정 데이터(다음)
    NEXT_BODY_DATA3 : WORD ;	//차종 설정 데이터(다음)
    NEXT_BODY_DATA4 : WORD ;	//차종 설정 데이터(다음)
    NEXT_RESERVED_DATA1 : WORD ;	//차종 설정 데이터(다음)
    NEXT_RESERVED_DATA2 : WORD ;	//차종 설정 데이터(다음)
    RESERVED4 : WORD ;
    RESERVED5 : WORD ;
   END_STRUCT ;
   FAC_Date_Time_DD_HH : WORD ;	//PLC 날짜,시간 보정을 위해 FAC가 주기적으로 날짜와 시간을 전송하는 영역
   FAC_Date_Time_MM_SS : WORD ;	//PLC 날짜,시간 보정을 위해 FAC가 주기적으로 분,초를 전송하는 영역
  END_STRUCT ;
BEGIN
   FAC1_IF.FAC_COMM_CHECK := 1;
   FAC1_IF.PLC_ONLINE_MODE := 0;
   FAC1_IF.STATION_WORK_COMPLETE := 0;
   FAC1_IF.PLC_DATA_REQ_COUNT := 1;
   FAC1_IF.FINAL_SEND_VINDATA1 := W#16#403;
   FAC1_IF.FINAL_SEND_VINDATA2 := W#16#2;
   FAC1_IF.RCV_DATA_CHECK_ERROR := 0;
   FAC1_IF.RESERVED1 := 0;
   FAC1_IF.RESERVED2 := 0;
   FAC1_IF.RESERVED3 := 0;
   FAC1_IF.LINE_DATA_READ_REQ := 11;
   FAC1_IF.ORDER_DATA_REQ := 1;
   FAC1_IF.PRESENT_VIN_DATA1 := W#16#0;
   FAC1_IF.PRESENT_VIN_DATA2 := W#16#0;
   FAC1_IF.PRESENT_BODY_DATA1 := W#16#0;
   FAC1_IF.PRESENT_BODY_DATA2 := W#16#0;
   FAC1_IF.PRESENT_BODY_DATA3 := W#16#0;
   FAC1_IF.PRESENT_BODY_DATA4 := W#16#0;
   FAC1_IF.PRESENT_RESERVED_DATA1 := W#16#0;
   FAC1_IF.PRESENT_RESERVED_DATA2 := W#16#0;
   FAC1_IF.NEXT_VIN_DATA1 := W#16#0;
   FAC1_IF.NEXT_VIN_DATA2 := W#16#0;
   FAC1_IF.NEXT_BODY_DATA1 := W#16#0;
   FAC1_IF.NEXT_BODY_DATA2 := W#16#0;
   FAC1_IF.NEXT_BODY_DATA3 := W#16#0;
   FAC1_IF.NEXT_BODY_DATA4 := W#16#0;
   FAC1_IF.NEXT_RESERVED_DATA1 := W#16#0;
   FAC1_IF.NEXT_RESERVED_DATA2 := W#16#0;
   FAC1_IF.RESERVED4 := W#16#0;
   FAC1_IF.RESERVED5 := W#16#0;
   FAC2_IF.FAC_COMM_CHECK := 1;
   FAC2_IF.PLC_ONLINE_MODE := 1;
   FAC2_IF.STATION_WORK_COMPLETE := 1;
   FAC2_IF.PLC_DATA_REQ_COUNT := 1;
   FAC2_IF.FINAL_SEND_VINDATA1 := W#16#4943;
   FAC2_IF.FINAL_SEND_VINDATA2 := W#16#23;
   FAC2_IF.RCV_DATA_CHECK_ERROR := 0;
   FAC2_IF.RESERVED1 := 0;
   FAC2_IF.RESERVED2 := 0;
   FAC2_IF.CMP_ORDER_DATA_REQ := 0;
   FAC2_IF.LINE_DATA_READ_REQ := 11;
   FAC2_IF.ORDER_DATA_REQ := 3;
   FAC2_IF.PRESENT_VIN_DATA1 := W#16#4943;
   FAC2_IF.PRESENT_VIN_DATA2 := W#16#23;
   FAC2_IF.PRESENT_BODY_DATA1 := W#16#4221;
   FAC2_IF.PRESENT_BODY_DATA := W#16#1080;
   FAC2_IF.PRESENT_BODY_DATA3 := W#16#562A;
   FAC2_IF.PRESENT_BODY_DATA4 := W#16#0;
   FAC2_IF.PRESENT_RESERVED_DATA1 := W#16#0;
   FAC2_IF.PRESENT_RESERVED_DATA2 := W#16#0;
   FAC2_IF.NEXT_VIN_DATA1 := W#16#4944;
   FAC2_IF.NEXT_VIN_DATA2 := W#16#23;
   FAC2_IF.NEXT_BODY_DATA1 := W#16#A21;
   FAC2_IF.NEXT_BODY_DATA2 := W#16#1040;
   FAC2_IF.NEXT_BODY_DATA3 := W#16#4616;
   FAC2_IF.NEXT_BODY_DATA4 := W#16#0;
   FAC2_IF.NEXT_RESERVED_DATA1 := W#16#0;
   FAC2_IF.NEXT_RESERVED_DATA2 := W#16#0;
   FAC2_IF.RESERVED4 := W#16#0;
   FAC2_IF.RESERVED5 := W#16#0;
   FAC3_IF.FAC_COMM_CHECK := 0;
   FAC3_IF.PLC_ONLINE_MODE := 0;
   FAC3_IF.STATION_WORK_COMPLETE := 0;
   FAC3_IF.PLC_DATA_REQ_COUNT := 0;
   FAC3_IF.FINAL_SEND_VINDATA1 := W#16#0;
   FAC3_IF.FINAL_SEND_VINDATA2 := W#16#0;
   FAC3_IF.RCV_DATA_CHECK_ERROR := 0;
   FAC3_IF.RESERVED1 := 0;
   FAC3_IF.RESERVED2 := 0;
   FAC3_IF.CMP_ORDER_DATA_REQ := 0;
   FAC3_IF.LINE_DATA_READ_REQ := 0;
   FAC3_IF.ORDER_DATA_REQ := 0;
   FAC3_IF.PRESENT_VIN_DATA1 := W#16#0;
   FAC3_IF.PRESENT_VIN_DATA2 := W#16#0;
   FAC3_IF.PRESENT_BODY_DATA1 := W#16#0;
   FAC3_IF.PRESENT_BODY_DATA := W#16#0;
   FAC3_IF.PRESENT_BODY_DATA3 := W#16#0;
   FAC3_IF.PRESENT_BODY_DATA4 := W#16#0;
   FAC3_IF.PRESENT_RESERVED_DATA1 := W#16#0;
   FAC3_IF.PRESENT_RESERVED_DATA2 := W#16#0;
   FAC3_IF.NEXT_VIN_DATA1 := W#16#0;
   FAC3_IF.NEXT_VIN_DATA2 := W#16#0;
   FAC3_IF.NEXT_BODY_DATA1 := W#16#0;
   FAC3_IF.NEXT_BODY_DATA2 := W#16#0;
   FAC3_IF.NEXT_BODY_DATA3 := W#16#0;
   FAC3_IF.NEXT_BODY_DATA4 := W#16#0;
   FAC3_IF.NEXT_RESERVED_DATA1 := W#16#0;
   FAC3_IF.NEXT_RESERVED_DATA2 := W#16#0;
   FAC3_IF.RESERVED4 := W#16#0;
   FAC3_IF.RESERVED5 := W#16#0;
   FAC4_IF.FAC_COMM_CHECK := 0;
   FAC4_IF.PLC_ONLINE_MODE := 0;
   FAC4_IF.STATION_WORK_COMPLETE := 0;
   FAC4_IF.PLC_DATA_REQ_COUNT := 0;
   FAC4_IF.FINAL_SEND_VINDATA1 := W#16#0;
   FAC4_IF.FINAL_SEND_VINDATA2 := W#16#0;
   FAC4_IF.RCV_DATA_CHECK_ERROR := 0;
   FAC4_IF.RESERVED1 := 0;
   FAC4_IF.RESERVED2 := 0;
   FAC4_IF.CMP_ORDER_DATA_REQ := 0;
   FAC4_IF.LINE_DATA_READ_REQ := 0;
   FAC4_IF.ORDER_DATA_REQ := 0;
   FAC4_IF.PRESENT_VIN_DATA1 := W#16#0;
   FAC4_IF.PRESENT_VIN_DATA2 := W#16#0;
   FAC4_IF.PRESENT_BODY_DATA1 := W#16#0;
   FAC4_IF.PRESENT_BODY_DATA := W#16#0;
   FAC4_IF.PRESENT_BODY_DATA3 := W#16#0;
   FAC4_IF.PRESENT_BODY_DATA4 := W#16#0;
   FAC4_IF.PRESENT_RESERVED_DATA1 := W#16#0;
   FAC4_IF.PRESENT_RESERVED_DATA2 := W#16#0;
   FAC4_IF.NEXT_VIN_DATA1 := W#16#0;
   FAC4_IF.NEXT_VIN_DATA2 := W#16#0;
   FAC4_IF.NEXT_BODY_DATA1 := W#16#0;
   FAC4_IF.NEXT_BODY_DATA2 := W#16#0;
   FAC4_IF.NEXT_BODY_DATA3 := W#16#0;
   FAC4_IF.NEXT_BODY_DATA4 := W#16#0;
   FAC4_IF.NEXT_RESERVED_DATA1 := W#16#0;
   FAC4_IF.NEXT_RESERVED_DATA2 := W#16#0;
   FAC4_IF.RESERVED4 := W#16#0;
   FAC4_IF.RESERVED5 := W#16#0;
   FAC5_IF.FAC_COMM_CHECK := 0;
   FAC5_IF.PLC_ONLINE_MODE := 0;
   FAC5_IF.STATION_WORK_COMPLETE := 0;
   FAC5_IF.PLC_DATA_REQ_COUNT := 0;
   FAC5_IF.FINAL_SEND_VINDATA1 := W#16#0;
   FAC5_IF.FINAL_SEND_VINDATA2 := W#16#0;
   FAC5_IF.RCV_DATA_CHECK_ERROR := 0;
   FAC5_IF.RESERVED1 := 0;
   FAC5_IF.RESERVED2 := 0;
   FAC5_IF.CMP_ORDER_DATA_REQ := 0;
   FAC5_IF.LINE_DATA_READ_REQ := 0;
   FAC5_IF.ORDER_DATA_REQ := 0;
   FAC5_IF.PRESENT_VIN_DATA1 := W#16#0;
   FAC5_IF.PRESENT_VIN_DATA2 := W#16#0;
   FAC5_IF.PRESENT_BODY_DATA1 := W#16#0;
   FAC5_IF.PRESENT_BODY_DATA := W#16#0;
   FAC5_IF.PRESENT_BODY_DATA3 := W#16#0;
   FAC5_IF.PRESENT_BODY_DATA4 := W#16#0;
   FAC5_IF.PRESENT_RESERVED_DATA1 := W#16#0;
   FAC5_IF.PRESENT_RESERVED_DATA2 := W#16#0;
   FAC5_IF.NEXT_VIN_DATA1 := W#16#0;
   FAC5_IF.NEXT_VIN_DATA2 := W#16#0;
   FAC5_IF.NEXT_BODY_DATA1 := W#16#0;
   FAC5_IF.NEXT_BODY_DATA2 := W#16#0;
   FAC5_IF.NEXT_BODY_DATA3 := W#16#0;
   FAC5_IF.NEXT_BODY_DATA4 := W#16#0;
   FAC5_IF.NEXT_RESERVED_DATA1 := W#16#0;
   FAC5_IF.NEXT_RESERVED_DATA2 := W#16#0;
   FAC5_IF.RESERVED4 := W#16#0;
   FAC5_IF.RESERVED5 := W#16#0;
   FAC6_IF.FAC_COMM_CHECK := 0;
   FAC6_IF.PLC_ONLINE_MODE := 0;
   FAC6_IF.STATION_WORK_COMPLETE := 0;
   FAC6_IF.PLC_DATA_REQ_COUNT := 0;
   FAC6_IF.FINAL_SEND_VINDATA1 := W#16#0;
   FAC6_IF.FINAL_SEND_VINDATA2 := W#16#0;
   FAC6_IF.RCV_DATA_CHECK_ERROR := 0;
   FAC6_IF.RESERVED1 := 0;
   FAC6_IF.RESERVED2 := 0;
   FAC6_IF.CMP_ORDER_DATA_REQ := 0;
   FAC6_IF.LINE_DATA_READ_REQ := 0;
   FAC6_IF.ORDER_DATA_REQ := 0;
   FAC6_IF.PRESENT_VIN_DATA1 := W#16#0;
   FAC6_IF.PRESENT_VIN_DATA2 := W#16#0;
   FAC6_IF.PRESENT_BODY_DATA1 := W#16#0;
   FAC6_IF.PRESENT_BODY_DATA := W#16#0;
   FAC6_IF.PRESENT_BODY_DATA3 := W#16#0;
   FAC6_IF.PRESENT_BODY_DATA4 := W#16#0;
   FAC6_IF.PRESENT_RESERVED_DATA1 := W#16#0;
   FAC6_IF.PRESENT_RESERVED_DATA2 := W#16#0;
   FAC6_IF.NEXT_VIN_DATA1 := W#16#0;
   FAC6_IF.NEXT_VIN_DATA2 := W#16#0;
   FAC6_IF.NEXT_BODY_DATA1 := W#16#0;
   FAC6_IF.NEXT_BODY_DATA2 := W#16#0;
   FAC6_IF.NEXT_BODY_DATA3 := W#16#0;
   FAC6_IF.NEXT_BODY_DATA4 := W#16#0;
   FAC6_IF.NEXT_RESERVED_DATA1 := W#16#0;
   FAC6_IF.NEXT_RESERVED_DATA2 := W#16#0;
   FAC6_IF.RESERVED4 := W#16#0;
   FAC6_IF.RESERVED5 := W#16#0;
   FAC7_IF.FAC_COMM_CHECK := 0;
   FAC7_IF.PLC_ONLINE_MODE := 0;
   FAC7_IF.STATION_WORK_COMPLETE := 0;
   FAC7_IF.PLC_DATA_REQ_COUNT := 0;
   FAC7_IF.FINAL_SEND_VINDATA1 := W#16#0;
   FAC7_IF.FINAL_SEND_VINDATA2 := W#16#0;
   FAC7_IF.RCV_DATA_CHECK_ERROR := 0;
   FAC7_IF.RESERVED1 := 0;
   FAC7_IF.RESERVED2 := 0;
   FAC7_IF.CMP_ORDER_DATA_REQ := 0;
   FAC7_IF.LINE_DATA_READ_REQ := 0;
   FAC7_IF.ORDER_DATA_REQ := 0;
   FAC7_IF.PRESENT_VIN_DATA1 := W#16#0;
   FAC7_IF.PRESENT_VIN_DATA2 := W#16#0;
   FAC7_IF.PRESENT_BODY_DATA1 := W#16#0;
   FAC7_IF.PRESENT_BODY_DATA := W#16#0;
   FAC7_IF.PRESENT_BODY_DATA3 := W#16#0;
   FAC7_IF.PRESENT_BODY_DATA4 := W#16#0;
   FAC7_IF.PRESENT_RESERVED_DATA1 := W#16#0;
   FAC7_IF.PRESENT_RESERVED_DATA2 := W#16#0;
   FAC7_IF.NEXT_VIN_DATA1 := W#16#0;
   FAC7_IF.NEXT_VIN_DATA2 := W#16#0;
   FAC7_IF.NEXT_BODY_DATA1 := W#16#0;
   FAC7_IF.NEXT_BODY_DATA2 := W#16#0;
   FAC7_IF.NEXT_BODY_DATA3 := W#16#0;
   FAC7_IF.NEXT_BODY_DATA4 := W#16#0;
   FAC7_IF.NEXT_RESERVED_DATA1 := W#16#0;
   FAC7_IF.NEXT_RESERVED_DATA2 := W#16#0;
   FAC7_IF.RESERVED4 := W#16#0;
   FAC7_IF.RESERVED5 := W#16#0;
   FAC8_IF.FAC_COMM_CHECK := 0;
   FAC8_IF.PLC_ONLINE_MODE := 0;
   FAC8_IF.STATION_WORK_COMPLETE := 0;
   FAC8_IF.PLC_DATA_REQ_COUNT := 0;
   FAC8_IF.FINAL_SEND_VINDATA1 := W#16#0;
   FAC8_IF.FINAL_SEND_VINDATA2 := W#16#0;
   FAC8_IF.RCV_DATA_CHECK_ERROR := 0;
   FAC8_IF.RESERVED1 := 0;
   FAC8_IF.RESERVED2 := 0;
   FAC8_IF.CMP_ORDER_DATA_REQ := 0;
   FAC8_IF.LINE_DATA_READ_REQ := 0;
   FAC8_IF.ORDER_DATA_REQ := 0;
   FAC8_IF.PRESENT_VIN_DATA1 := W#16#0;
   FAC8_IF.PRESENT_VIN_DATA2 := W#16#0;
   FAC8_IF.PRESENT_BODY_DATA1 := W#16#0;
   FAC8_IF.PRESENT_BODY_DATA := W#16#0;
   FAC8_IF.PRESENT_BODY_DATA3 := W#16#0;
   FAC8_IF.PRESENT_BODY_DATA4 := W#16#0;
   FAC8_IF.PRESENT_RESERVED_DATA1 := W#16#0;
   FAC8_IF.PRESENT_RESERVED_DATA2 := W#16#0;
   FAC8_IF.NEXT_VIN_DATA1 := W#16#0;
   FAC8_IF.NEXT_VIN_DATA2 := W#16#0;
   FAC8_IF.NEXT_BODY_DATA1 := W#16#0;
   FAC8_IF.NEXT_BODY_DATA2 := W#16#0;
   FAC8_IF.NEXT_BODY_DATA3 := W#16#0;
   FAC8_IF.NEXT_BODY_DATA4 := W#16#0;
   FAC8_IF.NEXT_RESERVED_DATA1 := W#16#0;
   FAC8_IF.NEXT_RESERVED_DATA2 := W#16#0;
   FAC8_IF.RESERVED4 := W#16#0;
   FAC8_IF.RESERVED5 := W#16#0;
   FAC9_IF.FAC_COMM_CHECK := 0;
   FAC9_IF.PLC_ONLINE_MODE := 0;
   FAC9_IF.STATION_WORK_COMPLETE := 0;
   FAC9_IF.PLC_DATA_REQ_COUNT := 0;
   FAC9_IF.FINAL_SEND_VINDATA1 := W#16#0;
   FAC9_IF.FINAL_SEND_VINDATA2 := W#16#0;
   FAC9_IF.RCV_DATA_CHECK_ERROR := 0;
   FAC9_IF.RESERVED1 := 0;
   FAC9_IF.RESERVED2 := 0;
   FAC9_IF.CMP_ORDER_DATA_REQ := 0;
   FAC9_IF.LINE_DATA_READ_REQ := 0;
   FAC9_IF.ORDER_DATA_REQ := 0;
   FAC9_IF.PRESENT_VIN_DATA1 := W#16#0;
   FAC9_IF.PRESENT_VIN_DATA2 := W#16#0;
   FAC9_IF.PRESENT_BODY_DATA1 := W#16#0;
   FAC9_IF.PRESENT_BODY_DATA := W#16#0;
   FAC9_IF.PRESENT_BODY_DATA3 := W#16#0;
   FAC9_IF.PRESENT_BODY_DATA4 := W#16#0;
   FAC9_IF.PRESENT_RESERVED_DATA1 := W#16#0;
   FAC9_IF.PRESENT_RESERVED_DATA2 := W#16#0;
   FAC9_IF.NEXT_VIN_DATA1 := W#16#0;
   FAC9_IF.NEXT_VIN_DATA2 := W#16#0;
   FAC9_IF.NEXT_BODY_DATA1 := W#16#0;
   FAC9_IF.NEXT_BODY_DATA2 := W#16#0;
   FAC9_IF.NEXT_BODY_DATA3 := W#16#0;
   FAC9_IF.NEXT_BODY_DATA4 := W#16#0;
   FAC9_IF.NEXT_RESERVED_DATA1 := W#16#0;
   FAC9_IF.NEXT_RESERVED_DATA2 := W#16#0;
   FAC9_IF.RESERVED4 := W#16#0;
   FAC9_IF.RESERVED5 := W#16#0;
   FAC10_IF.FAC_COMM_CHECK := 0;
   FAC10_IF.PLC_ONLINE_MODE := 0;
   FAC10_IF.STATION_WORK_COMPLETE := 0;
   FAC10_IF.PLC_DATA_REQ_COUNT := 0;
   FAC10_IF.FINAL_SEND_VINDATA1 := W#16#0;
   FAC10_IF.FINAL_SEND_VINDATA2 := W#16#0;
   FAC10_IF.RCV_DATA_CHECK_ERROR := 0;
   FAC10_IF.RESERVED1 := 0;
   FAC10_IF.RESERVED2 := 0;
   FAC10_IF.CMP_ORDER_DATA_REQ := 0;
   FAC10_IF.LINE_DATA_READ_REQ := 0;
   FAC10_IF.ORDER_DATA_REQ := 0;
   FAC10_IF.PRESENT_VIN_DATA1 := W#16#0;
   FAC10_IF.PRESENT_VIN_DATA2 := W#16#0;
   FAC10_IF.PRESENT_BODY_DATA1 := W#16#0;
   FAC10_IF.PRESENT_BODY_DATA := W#16#0;
   FAC10_IF.PRESENT_BODY_DATA3 := W#16#0;
   FAC10_IF.PRESENT_BODY_DATA4 := W#16#0;
   FAC10_IF.PRESENT_RESERVED_DATA1 := W#16#0;
   FAC10_IF.PRESENT_RESERVED_DATA2 := W#16#0;
   FAC10_IF.NEXT_VIN_DATA1 := W#16#0;
   FAC10_IF.NEXT_VIN_DATA2 := W#16#0;
   FAC10_IF.NEXT_BODY_DATA1 := W#16#0;
   FAC10_IF.NEXT_BODY_DATA2 := W#16#0;
   FAC10_IF.NEXT_BODY_DATA3 := W#16#0;
   FAC10_IF.NEXT_BODY_DATA4 := W#16#0;
   FAC10_IF.NEXT_RESERVED_DATA1 := W#16#0;
   FAC10_IF.NEXT_RESERVED_DATA2 := W#16#0;
   FAC10_IF.RESERVED4 := W#16#0;
   FAC10_IF.RESERVED5 := W#16#0;
   FAC11_IF.FAC_COMM_CHECK := 0;
   FAC11_IF.PLC_ONLINE_MODE := 0;
   FAC11_IF.STATION_WORK_COMPLETE := 0;
   FAC11_IF.PLC_DATA_REQ_COUNT := 0;
   FAC11_IF.FINAL_SEND_VINDATA1 := W#16#0;
   FAC11_IF.FINAL_SEND_VINDATA2 := W#16#0;
   FAC11_IF.RCV_DATA_CHECK_ERROR := 0;
   FAC11_IF.RESERVED1 := 0;
   FAC11_IF.RESERVED2 := 0;
   FAC11_IF.CMP_ORDER_DATA_REQ := 0;
   FAC11_IF.LINE_DATA_READ_REQ := 0;
   FAC11_IF.ORDER_DATA_REQ := 0;
   FAC11_IF.PRESENT_VIN_DATA1 := W#16#0;
   FAC11_IF.PRESENT_VIN_DATA2 := W#16#0;
   FAC11_IF.PRESENT_BODY_DATA1 := W#16#0;
   FAC11_IF.PRESENT_BODY_DATA := W#16#0;
   FAC11_IF.PRESENT_BODY_DATA3 := W#16#0;
   FAC11_IF.PRESENT_BODY_DATA4 := W#16#0;
   FAC11_IF.PRESENT_RESERVED_DATA1 := W#16#0;
   FAC11_IF.PRESENT_RESERVED_DATA2 := W#16#0;
   FAC11_IF.NEXT_VIN_DATA1 := W#16#0;
   FAC11_IF.NEXT_VIN_DATA2 := W#16#0;
   FAC11_IF.NEXT_BODY_DATA1 := W#16#0;
   FAC11_IF.NEXT_BODY_DATA2 := W#16#0;
   FAC11_IF.NEXT_BODY_DATA3 := W#16#0;
   FAC11_IF.NEXT_BODY_DATA4 := W#16#0;
   FAC11_IF.NEXT_RESERVED_DATA1 := W#16#0;
   FAC11_IF.NEXT_RESERVED_DATA2 := W#16#0;
   FAC11_IF.RESERVED4 := W#16#0;
   FAC11_IF.RESERVED5 := W#16#0;
   FAC12_IF.FAC_COMM_CHECK := 0;
   FAC12_IF.PLC_ONLINE_MODE := 0;
   FAC12_IF.STATION_WORK_COMPLETE := 0;
   FAC12_IF.PLC_DATA_REQ_COUNT := 0;
   FAC12_IF.FINAL_SEND_VINDATA1 := W#16#0;
   FAC12_IF.FINAL_SEND_VINDATA2 := W#16#0;
   FAC12_IF.RCV_DATA_CHECK_ERROR := 0;
   FAC12_IF.RESERVED1 := 0;
   FAC12_IF.RESERVED2 := 0;
   FAC12_IF.CMP_ORDER_DATA_REQ := 0;
   FAC12_IF.LINE_DATA_READ_REQ := 0;
   FAC12_IF.ORDER_DATA_REQ := 0;
   FAC12_IF.PRESENT_VIN_DATA1 := W#16#0;
   FAC12_IF.PRESENT_VIN_DATA2 := W#16#0;
   FAC12_IF.PRESENT_BODY_DATA1 := W#16#0;
   FAC12_IF.PRESENT_BODY_DATA := W#16#0;
   FAC12_IF.PRESENT_BODY_DATA3 := W#16#0;
   FAC12_IF.PRESENT_BODY_DATA4 := W#16#0;
   FAC12_IF.PRESENT_RESERVED_DATA1 := W#16#0;
   FAC12_IF.PRESENT_RESERVED_DATA2 := W#16#0;
   FAC12_IF.NEXT_VIN_DATA1 := W#16#0;
   FAC12_IF.NEXT_VIN_DATA2 := W#16#0;
   FAC12_IF.NEXT_BODY_DATA1 := W#16#0;
   FAC12_IF.NEXT_BODY_DATA2 := W#16#0;
   FAC12_IF.NEXT_BODY_DATA3 := W#16#0;
   FAC12_IF.NEXT_BODY_DATA4 := W#16#0;
   FAC12_IF.NEXT_RESERVED_DATA1 := W#16#0;
   FAC12_IF.NEXT_RESERVED_DATA2 := W#16#0;
   FAC12_IF.RESERVED4 := W#16#0;
   FAC12_IF.RESERVED5 := W#16#0;
   FAC13_IF.FAC_COMM_CHECK := 0;
   FAC13_IF.PLC_ONLINE_MODE := 0;
   FAC13_IF.STATION_WORK_COMPLETE := 0;
   FAC13_IF.PLC_DATA_REQ_COUNT := 0;
   FAC13_IF.FINAL_SEND_VINDATA1 := W#16#0;
   FAC13_IF.FINAL_SEND_VINDATA2 := W#16#0;
   FAC13_IF.RCV_DATA_CHECK_ERROR := 0;
   FAC13_IF.RESERVED1 := 0;
   FAC13_IF.RESERVED2 := 0;
   FAC13_IF.CMP_ORDER_DATA_REQ := 0;
   FAC13_IF.LINE_DATA_READ_REQ := 0;
   FAC13_IF.ORDER_DATA_REQ := 0;
   FAC13_IF.PRESENT_VIN_DATA1 := W#16#0;
   FAC13_IF.PRESENT_VIN_DATA2 := W#16#0;
   FAC13_IF.PRESENT_BODY_DATA1 := W#16#0;
   FAC13_IF.PRESENT_BODY_DATA := W#16#0;
   FAC13_IF.PRESENT_BODY_DATA3 := W#16#0;
   FAC13_IF.PRESENT_BODY_DATA4 := W#16#0;
   FAC13_IF.PRESENT_RESERVED_DATA1 := W#16#0;
   FAC13_IF.PRESENT_RESERVED_DATA2 := W#16#0;
   FAC13_IF.NEXT_VIN_DATA1 := W#16#0;
   FAC13_IF.NEXT_VIN_DATA2 := W#16#0;
   FAC13_IF.NEXT_BODY_DATA1 := W#16#0;
   FAC13_IF.NEXT_BODY_DATA2 := W#16#0;
   FAC13_IF.NEXT_BODY_DATA3 := W#16#0;
   FAC13_IF.NEXT_BODY_DATA4 := W#16#0;
   FAC13_IF.NEXT_RESERVED_DATA1 := W#16#0;
   FAC13_IF.NEXT_RESERVED_DATA2 := W#16#0;
   FAC13_IF.RESERVED4 := W#16#0;
   FAC13_IF.RESERVED5 := W#16#0;
   FAC14_IF.FAC_COMM_CHECK := 0;
   FAC14_IF.PLC_ONLINE_MODE := 0;
   FAC14_IF.STATION_WORK_COMPLETE := 0;
   FAC14_IF.PLC_DATA_REQ_COUNT := 0;
   FAC14_IF.FINAL_SEND_VINDATA1 := W#16#0;
   FAC14_IF.FINAL_SEND_VINDATA2 := W#16#0;
   FAC14_IF.RCV_DATA_CHECK_ERROR := 0;
   FAC14_IF.RESERVED1 := 0;
   FAC14_IF.RESERVED2 := 0;
   FAC14_IF.CMP_ORDER_DATA_REQ := 0;
   FAC14_IF.LINE_DATA_READ_REQ := 0;
   FAC14_IF.ORDER_DATA_REQ := 0;
   FAC14_IF.PRESENT_VIN_DATA1 := W#16#0;
   FAC14_IF.PRESENT_VIN_DATA2 := W#16#0;
   FAC14_IF.PRESENT_BODY_DATA1 := W#16#0;
   FAC14_IF.PRESENT_BODY_DATA := W#16#0;
   FAC14_IF.PRESENT_BODY_DATA3 := W#16#0;
   FAC14_IF.PRESENT_BODY_DATA4 := W#16#0;
   FAC14_IF.PRESENT_RESERVED_DATA1 := W#16#0;
   FAC14_IF.PRESENT_RESERVED_DATA2 := W#16#0;
   FAC14_IF.NEXT_VIN_DATA1 := W#16#0;
   FAC14_IF.NEXT_VIN_DATA2 := W#16#0;
   FAC14_IF.NEXT_BODY_DATA1 := W#16#0;
   FAC14_IF.NEXT_BODY_DATA2 := W#16#0;
   FAC14_IF.NEXT_BODY_DATA3 := W#16#0;
   FAC14_IF.NEXT_BODY_DATA4 := W#16#0;
   FAC14_IF.NEXT_RESERVED_DATA1 := W#16#0;
   FAC14_IF.NEXT_RESERVED_DATA2 := W#16#0;
   FAC14_IF.RESERVED4 := W#16#0;
   FAC14_IF.RESERVED5 := W#16#0;
   FAC15_IF.FAC_COMM_CHECK := 0;
   FAC15_IF.PLC_ONLINE_MODE := 0;
   FAC15_IF.STATION_WORK_COMPLETE := 0;
   FAC15_IF.PLC_DATA_REQ_COUNT := 0;
   FAC15_IF.FINAL_SEND_VINDATA1 := W#16#0;
   FAC15_IF.FINAL_SEND_VINDATA2 := W#16#0;
   FAC15_IF.RCV_DATA_CHECK_ERROR := 0;
   FAC15_IF.RESERVED1 := 0;
   FAC15_IF.RESERVED2 := 0;
   FAC15_IF.CMP_ORDER_DATA_REQ := 0;
   FAC15_IF.LINE_DATA_READ_REQ := 0;
   FAC15_IF.ORDER_DATA_REQ := 0;
   FAC15_IF.PRESENT_VIN_DATA1 := W#16#0;
   FAC15_IF.PRESENT_VIN_DATA2 := W#16#0;
   FAC15_IF.PRESENT_BODY_DATA1 := W#16#0;
   FAC15_IF.PRESENT_BODY_DATA := W#16#0;
   FAC15_IF.PRESENT_BODY_DATA3 := W#16#0;
   FAC15_IF.PRESENT_BODY_DATA4 := W#16#0;
   FAC15_IF.PRESENT_RESERVED_DATA1 := W#16#0;
   FAC15_IF.PRESENT_RESERVED_DATA2 := W#16#0;
   FAC15_IF.NEXT_VIN_DATA1 := W#16#0;
   FAC15_IF.NEXT_VIN_DATA2 := W#16#0;
   FAC15_IF.NEXT_BODY_DATA1 := W#16#0;
   FAC15_IF.NEXT_BODY_DATA2 := W#16#0;
   FAC15_IF.NEXT_BODY_DATA3 := W#16#0;
   FAC15_IF.NEXT_BODY_DATA4 := W#16#0;
   FAC15_IF.NEXT_RESERVED_DATA1 := W#16#0;
   FAC15_IF.NEXT_RESERVED_DATA2 := W#16#0;
   FAC15_IF.RESERVED4 := W#16#0;
   FAC15_IF.RESERVED5 := W#16#0;
   FAC16_IF.FAC_COMM_CHECK := 0;
   FAC16_IF.PLC_ONLINE_MODE := 0;
   FAC16_IF.STATION_WORK_COMPLETE := 0;
   FAC16_IF.PLC_DATA_REQ_COUNT := 0;
   FAC16_IF.FINAL_SEND_VINDATA1 := W#16#0;
   FAC16_IF.FINAL_SEND_VINDATA2 := W#16#0;
   FAC16_IF.RCV_DATA_CHECK_ERROR := 0;
   FAC16_IF.RESERVED1 := 0;
   FAC16_IF.RESERVED2 := 0;
   FAC16_IF.CMP_ORDER_DATA_REQ := 0;
   FAC16_IF.LINE_DATA_READ_REQ := 0;
   FAC16_IF.ORDER_DATA_REQ := 0;
   FAC16_IF.PRESENT_VIN_DATA1 := W#16#0;
   FAC16_IF.PRESENT_VIN_DATA2 := W#16#0;
   FAC16_IF.PRESENT_BODY_DATA1 := W#16#0;
   FAC16_IF.PRESENT_BODY_DATA := W#16#0;
   FAC16_IF.PRESENT_BODY_DATA3 := W#16#0;
   FAC16_IF.PRESENT_BODY_DATA4 := W#16#0;
   FAC16_IF.PRESENT_RESERVED_DATA1 := W#16#0;
   FAC16_IF.PRESENT_RESERVED_DATA2 := W#16#0;
   FAC16_IF.NEXT_VIN_DATA1 := W#16#0;
   FAC16_IF.NEXT_VIN_DATA2 := W#16#0;
   FAC16_IF.NEXT_BODY_DATA1 := W#16#0;
   FAC16_IF.NEXT_BODY_DATA2 := W#16#0;
   FAC16_IF.NEXT_BODY_DATA3 := W#16#0;
   FAC16_IF.NEXT_BODY_DATA4 := W#16#0;
   FAC16_IF.NEXT_RESERVED_DATA1 := W#16#0;
   FAC16_IF.NEXT_RESERVED_DATA2 := W#16#0;
   FAC16_IF.RESERVED4 := W#16#0;
   FAC16_IF.RESERVED5 := W#16#0;
   FAC_Date_Time_DD_HH := W#16#0;
   FAC_Date_Time_MM_SS := W#16#0;
END_DATA_BLOCK

DATA_BLOCK DB 161
TITLE =
VERSION : 0.1


  STRUCT
   Compare_VIN_Data1 : WORD ;	//수신 데이터 비교용 임시영역
   Compare_VIN_Data2 : WORD ;	//수신 데이터 비교용 임시영역
   Compare_Body_Data1 : WORD ;	//수신 데이터 비교용 임시영역
   Compare_Body_Data2 : WORD ;	//수신 데이터 비교용 임시영역
   Compare_Body_Data3 : WORD ;	//수신 데이터 비교용 임시영역
   Compare_Body_Data4 : WORD ;	//수신 데이터 비교용 임시영역
   Compare_Body_Data5 : WORD ;	//수신 데이터 비교용 임시영역
   Compare_Body_Data6 : WORD ;	//수신 데이터 비교용 임시영역
   Present_VIN_Data1 : WORD ;	//현재 공정 데이터 저장영역
   Present_VIN_Data2 : WORD ;	//현재 공정 데이터 저장영역
   Present_Body_Data1 : WORD ;	//현재 공정 데이터 저장영역
   Present_Body_Data2 : WORD ;	//현재 공정 데이터 저장영역
   Present_Body_Data3 : WORD ;	//현재 공정 데이터 저장영역
   Present_Body_Data4 : WORD ;	//현재 공정 데이터 저장영역
   Present_Body_Data5 : WORD ;	//현재 공정 데이터 저장영역
   Present_Body_Data6 : WORD ;	//현재 공정 데이터 저장영역
   Communication_Check1 : INT ;	//통신 확인용 1
   Communication_Check2 : INT ;	//통신 확인용 2
   FAC_IF_Data_OldValue : INT ;	//차종 설정 요청 정보 확인용 임시 저장 영역
   Data_REQ_Delay : INT ;
   Read_Date_Time : ARRAY  [1 .. 6 ] OF //PLC 현재 Date&Time Read 후 저장영역
   BYTE ;
   Set_Date_Time : ARRAY  [1 .. 6 ] OF //PLC Date&Time 변경 Data 저장영역
   BYTE ;
   Temporary_Bit : ARRAY  [1 .. 40 ] OF //생산지시용 함수 내부 사용 Bit Memory
   BOOL  := FALSE;
   Temporary_Bit_PLS : ARRAY  [1 .. 40 ] OF //생산지시용 함수 내부 사용 Pulse Bit Memory
   BOOL  := FALSE;
   unused2 : WORD ;
   unused3 : WORD ;
   unused4 : WORD ;
   unused5 : WORD ;
   unused6 : WORD ;
   unused7 : WORD ;
   unused8 : WORD ;
   Temporary : ARRAY  [1 .. 7 ] OF WORD ;
   LOG_LOOP_CNT : INT ;	//LOG저장시 루프 카운터값 저장
   LOG_LOOP_INDEX1 : INT ;	//LOG저장시 MOV포인트 기억용1
   LOG_LOOP_INDEX2 : INT ;	//LOG저장시 MOV포인트 기억용2
   TEMP_INT1 : INT ;
   LOG_STORE_DATA : ARRAY  [1 .. 500 ] OF //로그 저장 영역
   WORD ;
   ORDER_DATA_SWAP : ARRAY  [1 .. 16 ] OF BYTE ;
   TEMP1 : ARRAY  [1 .. 4 ] OF BYTE ;
   LINE_PRESENT_SWAP : ARRAY  [1 .. 16 ] OF BYTE ;
  END_STRUCT ;
BEGIN
   Compare_VIN_Data1 := W#16#0;
   Compare_VIN_Data2 := W#16#0;
   Compare_Body_Data1 := W#16#0;
   Compare_Body_Data2 := W#16#0;
   Compare_Body_Data3 := W#16#0;
   Compare_Body_Data4 := W#16#0;
   Compare_Body_Data5 := W#16#0;
   Compare_Body_Data6 := W#16#0;
   Present_VIN_Data1 := W#16#0;
   Present_VIN_Data2 := W#16#0;
   Present_Body_Data1 := W#16#0;
   Present_Body_Data2 := W#16#0;
   Present_Body_Data3 := W#16#0;
   Present_Body_Data4 := W#16#0;
   Present_Body_Data5 := W#16#0;
   Present_Body_Data6 := W#16#0;
   Communication_Check1 := 0;
   Communication_Check2 := 10;
   FAC_IF_Data_OldValue := 3;
   Data_REQ_Delay := 0;
   Read_Date_Time[1] := B#16#9;
   Read_Date_Time[2] := B#16#11;
   Read_Date_Time[3] := B#16#0;
   Read_Date_Time[4] := B#16#0;
   Read_Date_Time[5] := B#16#0;
   Read_Date_Time[6] := B#16#0;
   Set_Date_Time[1] := B#16#0;
   Set_Date_Time[2] := B#16#0;
   Set_Date_Time[3] := B#16#0;
   Set_Date_Time[4] := B#16#0;
   Set_Date_Time[5] := B#16#0;
   Set_Date_Time[6] := B#16#0;
   Temporary_Bit[1] := FALSE;
   Temporary_Bit[2] := FALSE;
   Temporary_Bit[3] := TRUE;
   Temporary_Bit[4] := FALSE;
   Temporary_Bit[5] := FALSE;
   Temporary_Bit[6] := FALSE;
   Temporary_Bit[7] := FALSE;
   Temporary_Bit[8] := FALSE;
   Temporary_Bit[9] := FALSE;
   Temporary_Bit[10] := FALSE;
   Temporary_Bit[11] := FALSE;
   Temporary_Bit[12] := FALSE;
   Temporary_Bit[13] := FALSE;
   Temporary_Bit[14] := FALSE;
   Temporary_Bit[15] := FALSE;
   Temporary_Bit[16] := FALSE;
   Temporary_Bit[17] := FALSE;
   Temporary_Bit[18] := FALSE;
   Temporary_Bit[19] := FALSE;
   Temporary_Bit[20] := FALSE;
   Temporary_Bit[21] := FALSE;
   Temporary_Bit[22] := FALSE;
   Temporary_Bit[23] := FALSE;
   Temporary_Bit[24] := FALSE;
   Temporary_Bit[25] := FALSE;
   Temporary_Bit[26] := FALSE;
   Temporary_Bit[27] := FALSE;
   Temporary_Bit[28] := FALSE;
   Temporary_Bit[29] := FALSE;
   Temporary_Bit[30] := FALSE;
   Temporary_Bit[31] := FALSE;
   Temporary_Bit[32] := FALSE;
   Temporary_Bit[33] := FALSE;
   Temporary_Bit[34] := FALSE;
   Temporary_Bit[35] := FALSE;
   Temporary_Bit[36] := FALSE;
   Temporary_Bit[37] := FALSE;
   Temporary_Bit[38] := FALSE;
   Temporary_Bit[39] := FALSE;
   Temporary_Bit[40] := FALSE;
   Temporary_Bit_PLS[1] := FALSE;
   Temporary_Bit_PLS[2] := FALSE;
   Temporary_Bit_PLS[3] := FALSE;
   Temporary_Bit_PLS[4] := FALSE;
   Temporary_Bit_PLS[5] := FALSE;
   Temporary_Bit_PLS[6] := TRUE;
   Temporary_Bit_PLS[7] := FALSE;
   Temporary_Bit_PLS[8] := TRUE;
   Temporary_Bit_PLS[9] := FALSE;
   Temporary_Bit_PLS[10] := FALSE;
   Temporary_Bit_PLS[11] := FALSE;
   Temporary_Bit_PLS[12] := FALSE;
   Temporary_Bit_PLS[13] := FALSE;
   Temporary_Bit_PLS[14] := FALSE;
   Temporary_Bit_PLS[15] := FALSE;
   Temporary_Bit_PLS[16] := FALSE;
   Temporary_Bit_PLS[17] := FALSE;
   Temporary_Bit_PLS[18] := FALSE;
   Temporary_Bit_PLS[19] := FALSE;
   Temporary_Bit_PLS[20] := FALSE;
   Temporary_Bit_PLS[21] := FALSE;
   Temporary_Bit_PLS[22] := FALSE;
   Temporary_Bit_PLS[23] := FALSE;
   Temporary_Bit_PLS[24] := FALSE;
   Temporary_Bit_PLS[25] := FALSE;
   Temporary_Bit_PLS[26] := FALSE;
   Temporary_Bit_PLS[27] := FALSE;
   Temporary_Bit_PLS[28] := FALSE;
   Temporary_Bit_PLS[29] := FALSE;
   Temporary_Bit_PLS[30] := FALSE;
   Temporary_Bit_PLS[31] := FALSE;
   Temporary_Bit_PLS[32] := FALSE;
   Temporary_Bit_PLS[33] := FALSE;
   Temporary_Bit_PLS[34] := FALSE;
   Temporary_Bit_PLS[35] := FALSE;
   Temporary_Bit_PLS[36] := FALSE;
   Temporary_Bit_PLS[37] := FALSE;
   Temporary_Bit_PLS[38] := FALSE;
   Temporary_Bit_PLS[39] := FALSE;
   Temporary_Bit_PLS[40] := FALSE;
   unused2 := W#16#0;
   unused3 := W#16#0;
   unused4 := W#16#0;
   unused5 := W#16#0;
   unused6 := W#16#0;
   unused7 := W#16#0;
   unused8 := W#16#0;
   Temporary[1] := W#16#0;
   Temporary[2] := W#16#0;
   Temporary[3] := W#16#0;
   Temporary[4] := W#16#0;
   Temporary[5] := W#16#0;
   Temporary[6] := W#16#0;
   Temporary[7] := W#16#0;
   LOG_LOOP_CNT := 100;
   LOG_LOOP_INDEX1 := 90;
   LOG_LOOP_INDEX2 := 80;
   TEMP_INT1 := 0;
   LOG_STORE_DATA[1] := W#16#500;
   LOG_STORE_DATA[2] := W#16#1312;
   LOG_STORE_DATA[3] := W#16#1;
   LOG_STORE_DATA[4] := W#16#0;
   LOG_STORE_DATA[5] := W#16#0;
   LOG_STORE_DATA[6] := W#16#400;
   LOG_STORE_DATA[7] := W#16#1311;
   LOG_STORE_DATA[8] := W#16#5950;
   LOG_STORE_DATA[9] := W#16#0;
   LOG_STORE_DATA[10] := W#16#0;
   LOG_STORE_DATA[11] := W#16#500;
   LOG_STORE_DATA[12] := W#16#1311;
   LOG_STORE_DATA[13] := W#16#5918;
   LOG_STORE_DATA[14] := W#16#0;
   LOG_STORE_DATA[15] := W#16#0;
   LOG_STORE_DATA[16] := W#16#400;
   LOG_STORE_DATA[17] := W#16#1311;
   LOG_STORE_DATA[18] := W#16#5907;
   LOG_STORE_DATA[19] := W#16#0;
   LOG_STORE_DATA[20] := W#16#0;
   LOG_STORE_DATA[21] := W#16#500;
   LOG_STORE_DATA[22] := W#16#1311;
   LOG_STORE_DATA[23] := W#16#4514;
   LOG_STORE_DATA[24] := W#16#0;
   LOG_STORE_DATA[25] := W#16#0;
   LOG_STORE_DATA[26] := W#16#400;
   LOG_STORE_DATA[27] := W#16#1311;
   LOG_STORE_DATA[28] := W#16#4504;
   LOG_STORE_DATA[29] := W#16#0;
   LOG_STORE_DATA[30] := W#16#0;
   LOG_STORE_DATA[31] := W#16#500;
   LOG_STORE_DATA[32] := W#16#1311;
   LOG_STORE_DATA[33] := W#16#4158;
   LOG_STORE_DATA[34] := W#16#0;
   LOG_STORE_DATA[35] := W#16#0;
   LOG_STORE_DATA[36] := W#16#400;
   LOG_STORE_DATA[37] := W#16#1311;
   LOG_STORE_DATA[38] := W#16#4148;
   LOG_STORE_DATA[39] := W#16#0;
   LOG_STORE_DATA[40] := W#16#0;
   LOG_STORE_DATA[41] := W#16#500;
   LOG_STORE_DATA[42] := W#16#1311;
   LOG_STORE_DATA[43] := W#16#4024;
   LOG_STORE_DATA[44] := W#16#0;
   LOG_STORE_DATA[45] := W#16#0;
   LOG_STORE_DATA[46] := W#16#400;
   LOG_STORE_DATA[47] := W#16#1311;
   LOG_STORE_DATA[48] := W#16#4014;
   LOG_STORE_DATA[49] := W#16#0;
   LOG_STORE_DATA[50] := W#16#0;
   LOG_STORE_DATA[51] := W#16#200;
   LOG_STORE_DATA[52] := W#16#1311;
   LOG_STORE_DATA[53] := W#16#3722;
   LOG_STORE_DATA[54] := W#16#1;
   LOG_STORE_DATA[55] := W#16#403;
   LOG_STORE_DATA[56] := W#16#500;
   LOG_STORE_DATA[57] := W#16#1311;
   LOG_STORE_DATA[58] := W#16#3704;
   LOG_STORE_DATA[59] := W#16#0;
   LOG_STORE_DATA[60] := W#16#0;
   LOG_STORE_DATA[61] := W#16#400;
   LOG_STORE_DATA[62] := W#16#1311;
   LOG_STORE_DATA[63] := W#16#3654;
   LOG_STORE_DATA[64] := W#16#0;
   LOG_STORE_DATA[65] := W#16#0;
   LOG_STORE_DATA[66] := W#16#300;
   LOG_STORE_DATA[67] := W#16#1311;
   LOG_STORE_DATA[68] := W#16#3452;
   LOG_STORE_DATA[69] := W#16#B;
   LOG_STORE_DATA[70] := W#16#403;
   LOG_STORE_DATA[71] := W#16#200;
   LOG_STORE_DATA[72] := W#16#1311;
   LOG_STORE_DATA[73] := W#16#3451;
   LOG_STORE_DATA[74] := W#16#1;
   LOG_STORE_DATA[75] := W#16#386;
   LOG_STORE_DATA[76] := W#16#300;
   LOG_STORE_DATA[77] := W#16#1311;
   LOG_STORE_DATA[78] := W#16#3420;
   LOG_STORE_DATA[79] := W#16#B;
   LOG_STORE_DATA[80] := W#16#402;
   LOG_STORE_DATA[81] := W#16#500;
   LOG_STORE_DATA[82] := W#16#1311;
   LOG_STORE_DATA[83] := W#16#3413;
   LOG_STORE_DATA[84] := W#16#0;
   LOG_STORE_DATA[85] := W#16#0;
   LOG_STORE_DATA[86] := W#16#400;
   LOG_STORE_DATA[87] := W#16#1311;
   LOG_STORE_DATA[88] := W#16#3403;
   LOG_STORE_DATA[89] := W#16#0;
   LOG_STORE_DATA[90] := W#16#0;
   LOG_STORE_DATA[91] := W#16#200;
   LOG_STORE_DATA[92] := W#16#1311;
   LOG_STORE_DATA[93] := W#16#3341;
   LOG_STORE_DATA[94] := W#16#1;
   LOG_STORE_DATA[95] := W#16#386;
   LOG_STORE_DATA[96] := W#16#500;
   LOG_STORE_DATA[97] := W#16#1311;
   LOG_STORE_DATA[98] := W#16#3233;
   LOG_STORE_DATA[99] := W#16#0;
   LOG_STORE_DATA[100] := W#16#0;
   LOG_STORE_DATA[101] := W#16#600;
   LOG_STORE_DATA[102] := W#16#1311;
   LOG_STORE_DATA[103] := W#16#3229;
   LOG_STORE_DATA[104] := W#16#64;
   LOG_STORE_DATA[105] := W#16#401;
   LOG_STORE_DATA[106] := W#16#400;
   LOG_STORE_DATA[107] := W#16#1311;
   LOG_STORE_DATA[108] := W#16#3222;
   LOG_STORE_DATA[109] := W#16#0;
   LOG_STORE_DATA[110] := W#16#0;
   LOG_STORE_DATA[111] := W#16#300;
   LOG_STORE_DATA[112] := W#16#1311;
   LOG_STORE_DATA[113] := W#16#3202;
   LOG_STORE_DATA[114] := W#16#B;
   LOG_STORE_DATA[115] := W#16#400;
   LOG_STORE_DATA[116] := W#16#200;
   LOG_STORE_DATA[117] := W#16#1311;
   LOG_STORE_DATA[118] := W#16#3201;
   LOG_STORE_DATA[119] := W#16#1;
   LOG_STORE_DATA[120] := W#16#386;
   LOG_STORE_DATA[121] := W#16#300;
   LOG_STORE_DATA[122] := W#16#1311;
   LOG_STORE_DATA[123] := W#16#3145;
   LOG_STORE_DATA[124] := W#16#B;
   LOG_STORE_DATA[125] := W#16#399;
   LOG_STORE_DATA[126] := W#16#500;
   LOG_STORE_DATA[127] := W#16#1311;
   LOG_STORE_DATA[128] := W#16#3119;
   LOG_STORE_DATA[129] := W#16#0;
   LOG_STORE_DATA[130] := W#16#0;
   LOG_STORE_DATA[131] := W#16#400;
   LOG_STORE_DATA[132] := W#16#1311;
   LOG_STORE_DATA[133] := W#16#3109;
   LOG_STORE_DATA[134] := W#16#0;
   LOG_STORE_DATA[135] := W#16#0;
   LOG_STORE_DATA[136] := W#16#500;
   LOG_STORE_DATA[137] := W#16#1311;
   LOG_STORE_DATA[138] := W#16#2958;
   LOG_STORE_DATA[139] := W#16#0;
   LOG_STORE_DATA[140] := W#16#0;
   LOG_STORE_DATA[141] := W#16#400;
   LOG_STORE_DATA[142] := W#16#1311;
   LOG_STORE_DATA[143] := W#16#2947;
   LOG_STORE_DATA[144] := W#16#0;
   LOG_STORE_DATA[145] := W#16#0;
   LOG_STORE_DATA[146] := W#16#200;
   LOG_STORE_DATA[147] := W#16#1311;
   LOG_STORE_DATA[148] := W#16#2926;
   LOG_STORE_DATA[149] := W#16#1;
   LOG_STORE_DATA[150] := W#16#386;
   LOG_STORE_DATA[151] := W#16#500;
   LOG_STORE_DATA[152] := W#16#1311;
   LOG_STORE_DATA[153] := W#16#2843;
   LOG_STORE_DATA[154] := W#16#0;
   LOG_STORE_DATA[155] := W#16#0;
   LOG_STORE_DATA[156] := W#16#400;
   LOG_STORE_DATA[157] := W#16#1311;
   LOG_STORE_DATA[158] := W#16#2833;
   LOG_STORE_DATA[159] := W#16#0;
   LOG_STORE_DATA[160] := W#16#0;
   LOG_STORE_DATA[161] := W#16#300;
   LOG_STORE_DATA[162] := W#16#1311;
   LOG_STORE_DATA[163] := W#16#2811;
   LOG_STORE_DATA[164] := W#16#B;
   LOG_STORE_DATA[165] := W#16#398;
   LOG_STORE_DATA[166] := W#16#200;
   LOG_STORE_DATA[167] := W#16#1311;
   LOG_STORE_DATA[168] := W#16#2810;
   LOG_STORE_DATA[169] := W#16#1;
   LOG_STORE_DATA[170] := W#16#386;
   LOG_STORE_DATA[171] := W#16#500;
   LOG_STORE_DATA[172] := W#16#1311;
   LOG_STORE_DATA[173] := W#16#2724;
   LOG_STORE_DATA[174] := W#16#0;
   LOG_STORE_DATA[175] := W#16#0;
   LOG_STORE_DATA[176] := W#16#400;
   LOG_STORE_DATA[177] := W#16#1311;
   LOG_STORE_DATA[178] := W#16#2714;
   LOG_STORE_DATA[179] := W#16#0;
   LOG_STORE_DATA[180] := W#16#0;
   LOG_STORE_DATA[181] := W#16#300;
   LOG_STORE_DATA[182] := W#16#1311;
   LOG_STORE_DATA[183] := W#16#2655;
   LOG_STORE_DATA[184] := W#16#B;
   LOG_STORE_DATA[185] := W#16#397;
   LOG_STORE_DATA[186] := W#16#200;
   LOG_STORE_DATA[187] := W#16#1311;
   LOG_STORE_DATA[188] := W#16#2653;
   LOG_STORE_DATA[189] := W#16#1;
   LOG_STORE_DATA[190] := W#16#386;
   LOG_STORE_DATA[191] := W#16#500;
   LOG_STORE_DATA[192] := W#16#1311;
   LOG_STORE_DATA[193] := W#16#2605;
   LOG_STORE_DATA[194] := W#16#0;
   LOG_STORE_DATA[195] := W#16#0;
   LOG_STORE_DATA[196] := W#16#400;
   LOG_STORE_DATA[197] := W#16#1311;
   LOG_STORE_DATA[198] := W#16#2554;
   LOG_STORE_DATA[199] := W#16#0;
   LOG_STORE_DATA[200] := W#16#0;
   LOG_STORE_DATA[201] := W#16#300;
   LOG_STORE_DATA[202] := W#16#1311;
   LOG_STORE_DATA[203] := W#16#2532;
   LOG_STORE_DATA[204] := W#16#B;
   LOG_STORE_DATA[205] := W#16#396;
   LOG_STORE_DATA[206] := W#16#200;
   LOG_STORE_DATA[207] := W#16#1311;
   LOG_STORE_DATA[208] := W#16#2531;
   LOG_STORE_DATA[209] := W#16#1;
   LOG_STORE_DATA[210] := W#16#386;
   LOG_STORE_DATA[211] := W#16#500;
   LOG_STORE_DATA[212] := W#16#1311;
   LOG_STORE_DATA[213] := W#16#2450;
   LOG_STORE_DATA[214] := W#16#0;
   LOG_STORE_DATA[215] := W#16#0;
   LOG_STORE_DATA[216] := W#16#600;
   LOG_STORE_DATA[217] := W#16#1311;
   LOG_STORE_DATA[218] := W#16#2441;
   LOG_STORE_DATA[219] := W#16#64;
   LOG_STORE_DATA[220] := W#16#395;
   LOG_STORE_DATA[221] := W#16#400;
   LOG_STORE_DATA[222] := W#16#1311;
   LOG_STORE_DATA[223] := W#16#2440;
   LOG_STORE_DATA[224] := W#16#0;
   LOG_STORE_DATA[225] := W#16#0;
   LOG_STORE_DATA[226] := W#16#300;
   LOG_STORE_DATA[227] := W#16#1311;
   LOG_STORE_DATA[228] := W#16#2414;
   LOG_STORE_DATA[229] := W#16#B;
   LOG_STORE_DATA[230] := W#16#394;
   LOG_STORE_DATA[231] := W#16#200;
   LOG_STORE_DATA[232] := W#16#1311;
   LOG_STORE_DATA[233] := W#16#2412;
   LOG_STORE_DATA[234] := W#16#1;
   LOG_STORE_DATA[235] := W#16#386;
   LOG_STORE_DATA[236] := W#16#500;
   LOG_STORE_DATA[237] := W#16#1311;
   LOG_STORE_DATA[238] := W#16#2331;
   LOG_STORE_DATA[239] := W#16#0;
   LOG_STORE_DATA[240] := W#16#0;
   LOG_STORE_DATA[241] := W#16#400;
   LOG_STORE_DATA[242] := W#16#1311;
   LOG_STORE_DATA[243] := W#16#2321;
   LOG_STORE_DATA[244] := W#16#0;
   LOG_STORE_DATA[245] := W#16#0;
   LOG_STORE_DATA[246] := W#16#600;
   LOG_STORE_DATA[247] := W#16#1311;
   LOG_STORE_DATA[248] := W#16#2224;
   LOG_STORE_DATA[249] := W#16#64;
   LOG_STORE_DATA[250] := W#16#393;
   LOG_STORE_DATA[251] := W#16#500;
   LOG_STORE_DATA[252] := W#16#1311;
   LOG_STORE_DATA[253] := W#16#2211;
   LOG_STORE_DATA[254] := W#16#0;
   LOG_STORE_DATA[255] := W#16#0;
   LOG_STORE_DATA[256] := W#16#400;
   LOG_STORE_DATA[257] := W#16#1311;
   LOG_STORE_DATA[258] := W#16#2201;
   LOG_STORE_DATA[259] := W#16#0;
   LOG_STORE_DATA[260] := W#16#0;
   LOG_STORE_DATA[261] := W#16#300;
   LOG_STORE_DATA[262] := W#16#1311;
   LOG_STORE_DATA[263] := W#16#2101;
   LOG_STORE_DATA[264] := W#16#B;
   LOG_STORE_DATA[265] := W#16#388;
   LOG_STORE_DATA[266] := W#16#200;
   LOG_STORE_DATA[267] := W#16#1311;
   LOG_STORE_DATA[268] := W#16#2059;
   LOG_STORE_DATA[269] := W#16#1;
   LOG_STORE_DATA[270] := W#16#386;
   LOG_STORE_DATA[271] := W#16#500;
   LOG_STORE_DATA[272] := W#16#1311;
   LOG_STORE_DATA[273] := W#16#2038;
   LOG_STORE_DATA[274] := W#16#0;
   LOG_STORE_DATA[275] := W#16#0;
   LOG_STORE_DATA[276] := W#16#400;
   LOG_STORE_DATA[277] := W#16#1311;
   LOG_STORE_DATA[278] := W#16#2027;
   LOG_STORE_DATA[279] := W#16#0;
   LOG_STORE_DATA[280] := W#16#0;
   LOG_STORE_DATA[281] := W#16#300;
   LOG_STORE_DATA[282] := W#16#1311;
   LOG_STORE_DATA[283] := W#16#2003;
   LOG_STORE_DATA[284] := W#16#B;
   LOG_STORE_DATA[285] := W#16#387;
   LOG_STORE_DATA[286] := W#16#500;
   LOG_STORE_DATA[287] := W#16#1311;
   LOG_STORE_DATA[288] := W#16#1925;
   LOG_STORE_DATA[289] := W#16#0;
   LOG_STORE_DATA[290] := W#16#0;
   LOG_STORE_DATA[291] := W#16#400;
   LOG_STORE_DATA[292] := W#16#1311;
   LOG_STORE_DATA[293] := W#16#1915;
   LOG_STORE_DATA[294] := W#16#0;
   LOG_STORE_DATA[295] := W#16#0;
   LOG_STORE_DATA[296] := W#16#500;
   LOG_STORE_DATA[297] := W#16#1311;
   LOG_STORE_DATA[298] := W#16#1807;
   LOG_STORE_DATA[299] := W#16#0;
   LOG_STORE_DATA[300] := W#16#0;
   LOG_STORE_DATA[301] := W#16#400;
   LOG_STORE_DATA[302] := W#16#1311;
   LOG_STORE_DATA[303] := W#16#1756;
   LOG_STORE_DATA[304] := W#16#0;
   LOG_STORE_DATA[305] := W#16#0;
   LOG_STORE_DATA[306] := W#16#500;
   LOG_STORE_DATA[307] := W#16#1311;
   LOG_STORE_DATA[308] := W#16#1646;
   LOG_STORE_DATA[309] := W#16#0;
   LOG_STORE_DATA[310] := W#16#0;
   LOG_STORE_DATA[311] := W#16#400;
   LOG_STORE_DATA[312] := W#16#1311;
   LOG_STORE_DATA[313] := W#16#1636;
   LOG_STORE_DATA[314] := W#16#0;
   LOG_STORE_DATA[315] := W#16#0;
   LOG_STORE_DATA[316] := W#16#500;
   LOG_STORE_DATA[317] := W#16#1311;
   LOG_STORE_DATA[318] := W#16#1452;
   LOG_STORE_DATA[319] := W#16#0;
   LOG_STORE_DATA[320] := W#16#0;
   LOG_STORE_DATA[321] := W#16#400;
   LOG_STORE_DATA[322] := W#16#1311;
   LOG_STORE_DATA[323] := W#16#1442;
   LOG_STORE_DATA[324] := W#16#0;
   LOG_STORE_DATA[325] := W#16#0;
   LOG_STORE_DATA[326] := W#16#500;
   LOG_STORE_DATA[327] := W#16#1311;
   LOG_STORE_DATA[328] := W#16#1241;
   LOG_STORE_DATA[329] := W#16#0;
   LOG_STORE_DATA[330] := W#16#0;
   LOG_STORE_DATA[331] := W#16#400;
   LOG_STORE_DATA[332] := W#16#1311;
   LOG_STORE_DATA[333] := W#16#1230;
   LOG_STORE_DATA[334] := W#16#0;
   LOG_STORE_DATA[335] := W#16#0;
   LOG_STORE_DATA[336] := W#16#200;
   LOG_STORE_DATA[337] := W#16#1311;
   LOG_STORE_DATA[338] := W#16#1034;
   LOG_STORE_DATA[339] := W#16#1;
   LOG_STORE_DATA[340] := W#16#386;
   LOG_STORE_DATA[341] := W#16#500;
   LOG_STORE_DATA[342] := W#16#1311;
   LOG_STORE_DATA[343] := W#16#947;
   LOG_STORE_DATA[344] := W#16#0;
   LOG_STORE_DATA[345] := W#16#0;
   LOG_STORE_DATA[346] := W#16#400;
   LOG_STORE_DATA[347] := W#16#1311;
   LOG_STORE_DATA[348] := W#16#937;
   LOG_STORE_DATA[349] := W#16#0;
   LOG_STORE_DATA[350] := W#16#0;
   LOG_STORE_DATA[351] := W#16#600;
   LOG_STORE_DATA[352] := W#16#1311;
   LOG_STORE_DATA[353] := W#16#908;
   LOG_STORE_DATA[354] := W#16#64;
   LOG_STORE_DATA[355] := W#16#386;
   LOG_STORE_DATA[356] := W#16#200;
   LOG_STORE_DATA[357] := W#16#1311;
   LOG_STORE_DATA[358] := W#16#900;
   LOG_STORE_DATA[359] := W#16#1;
   LOG_STORE_DATA[360] := W#16#383;
   LOG_STORE_DATA[361] := W#16#500;
   LOG_STORE_DATA[362] := W#16#1311;
   LOG_STORE_DATA[363] := W#16#837;
   LOG_STORE_DATA[364] := W#16#0;
   LOG_STORE_DATA[365] := W#16#0;
   LOG_STORE_DATA[366] := W#16#400;
   LOG_STORE_DATA[367] := W#16#1311;
   LOG_STORE_DATA[368] := W#16#827;
   LOG_STORE_DATA[369] := W#16#0;
   LOG_STORE_DATA[370] := W#16#0;
   LOG_STORE_DATA[371] := W#16#300;
   LOG_STORE_DATA[372] := W#16#1311;
   LOG_STORE_DATA[373] := W#16#819;
   LOG_STORE_DATA[374] := W#16#B;
   LOG_STORE_DATA[375] := W#16#384;
   LOG_STORE_DATA[376] := W#16#500;
   LOG_STORE_DATA[377] := W#16#1311;
   LOG_STORE_DATA[378] := W#16#706;
   LOG_STORE_DATA[379] := W#16#0;
   LOG_STORE_DATA[380] := W#16#0;
   LOG_STORE_DATA[381] := W#16#400;
   LOG_STORE_DATA[382] := W#16#1311;
   LOG_STORE_DATA[383] := W#16#656;
   LOG_STORE_DATA[384] := W#16#0;
   LOG_STORE_DATA[385] := W#16#0;
   LOG_STORE_DATA[386] := W#16#200;
   LOG_STORE_DATA[387] := W#16#1311;
   LOG_STORE_DATA[388] := W#16#416;
   LOG_STORE_DATA[389] := W#16#1;
   LOG_STORE_DATA[390] := W#16#383;
   LOG_STORE_DATA[391] := W#16#500;
   LOG_STORE_DATA[392] := W#16#1311;
   LOG_STORE_DATA[393] := W#16#340;
   LOG_STORE_DATA[394] := W#16#0;
   LOG_STORE_DATA[395] := W#16#0;
   LOG_STORE_DATA[396] := W#16#400;
   LOG_STORE_DATA[397] := W#16#1311;
   LOG_STORE_DATA[398] := W#16#330;
   LOG_STORE_DATA[399] := W#16#0;
   LOG_STORE_DATA[400] := W#16#0;
   LOG_STORE_DATA[401] := W#16#300;
   LOG_STORE_DATA[402] := W#16#1311;
   LOG_STORE_DATA[403] := W#16#306;
   LOG_STORE_DATA[404] := W#16#B;
   LOG_STORE_DATA[405] := W#16#383;
   LOG_STORE_DATA[406] := W#16#200;
   LOG_STORE_DATA[407] := W#16#1311;
   LOG_STORE_DATA[408] := W#16#246;
   LOG_STORE_DATA[409] := W#16#1;
   LOG_STORE_DATA[410] := W#16#382;
   LOG_STORE_DATA[411] := W#16#500;
   LOG_STORE_DATA[412] := W#16#1311;
   LOG_STORE_DATA[413] := W#16#235;
   LOG_STORE_DATA[414] := W#16#0;
   LOG_STORE_DATA[415] := W#16#0;
   LOG_STORE_DATA[416] := W#16#400;
   LOG_STORE_DATA[417] := W#16#1311;
   LOG_STORE_DATA[418] := W#16#225;
   LOG_STORE_DATA[419] := W#16#0;
   LOG_STORE_DATA[420] := W#16#0;
   LOG_STORE_DATA[421] := W#16#300;
   LOG_STORE_DATA[422] := W#16#1311;
   LOG_STORE_DATA[423] := W#16#147;
   LOG_STORE_DATA[424] := W#16#B;
   LOG_STORE_DATA[425] := W#16#382;
   LOG_STORE_DATA[426] := W#16#200;
   LOG_STORE_DATA[427] := W#16#1311;
   LOG_STORE_DATA[428] := W#16#136;
   LOG_STORE_DATA[429] := W#16#1;
   LOG_STORE_DATA[430] := W#16#381;
   LOG_STORE_DATA[431] := W#16#500;
   LOG_STORE_DATA[432] := W#16#1311;
   LOG_STORE_DATA[433] := W#16#55;
   LOG_STORE_DATA[434] := W#16#0;
   LOG_STORE_DATA[435] := W#16#0;
   LOG_STORE_DATA[436] := W#16#400;
   LOG_STORE_DATA[437] := W#16#1311;
   LOG_STORE_DATA[438] := W#16#44;
   LOG_STORE_DATA[439] := W#16#0;
   LOG_STORE_DATA[440] := W#16#0;
   LOG_STORE_DATA[441] := W#16#300;
   LOG_STORE_DATA[442] := W#16#1311;
   LOG_STORE_DATA[443] := W#16#31;
   LOG_STORE_DATA[444] := W#16#B;
   LOG_STORE_DATA[445] := W#16#381;
   LOG_STORE_DATA[446] := W#16#200;
   LOG_STORE_DATA[447] := W#16#1310;
   LOG_STORE_DATA[448] := W#16#5835;
   LOG_STORE_DATA[449] := W#16#1;
   LOG_STORE_DATA[450] := W#16#380;
   LOG_STORE_DATA[451] := W#16#500;
   LOG_STORE_DATA[452] := W#16#1310;
   LOG_STORE_DATA[453] := W#16#5806;
   LOG_STORE_DATA[454] := W#16#0;
   LOG_STORE_DATA[455] := W#16#0;
   LOG_STORE_DATA[456] := W#16#400;
   LOG_STORE_DATA[457] := W#16#1310;
   LOG_STORE_DATA[458] := W#16#5755;
   LOG_STORE_DATA[459] := W#16#0;
   LOG_STORE_DATA[460] := W#16#0;
   LOG_STORE_DATA[461] := W#16#300;
   LOG_STORE_DATA[462] := W#16#1310;
   LOG_STORE_DATA[463] := W#16#5722;
   LOG_STORE_DATA[464] := W#16#B;
   LOG_STORE_DATA[465] := W#16#380;
   LOG_STORE_DATA[466] := W#16#200;
   LOG_STORE_DATA[467] := W#16#1310;
   LOG_STORE_DATA[468] := W#16#5720;
   LOG_STORE_DATA[469] := W#16#1;
   LOG_STORE_DATA[470] := W#16#379;
   LOG_STORE_DATA[471] := W#16#500;
   LOG_STORE_DATA[472] := W#16#1310;
   LOG_STORE_DATA[473] := W#16#5654;
   LOG_STORE_DATA[474] := W#16#0;
   LOG_STORE_DATA[475] := W#16#0;
   LOG_STORE_DATA[476] := W#16#400;
   LOG_STORE_DATA[477] := W#16#1310;
   LOG_STORE_DATA[478] := W#16#5644;
   LOG_STORE_DATA[479] := W#16#0;
   LOG_STORE_DATA[480] := W#16#0;
   LOG_STORE_DATA[481] := W#16#300;
   LOG_STORE_DATA[482] := W#16#1310;
   LOG_STORE_DATA[483] := W#16#5556;
   LOG_STORE_DATA[484] := W#16#B;
   LOG_STORE_DATA[485] := W#16#379;
   LOG_STORE_DATA[486] := W#16#200;
   LOG_STORE_DATA[487] := W#16#1310;
   LOG_STORE_DATA[488] := W#16#5554;
   LOG_STORE_DATA[489] := W#16#1;
   LOG_STORE_DATA[490] := W#16#378;
   LOG_STORE_DATA[491] := W#16#500;
   LOG_STORE_DATA[492] := W#16#1310;
   LOG_STORE_DATA[493] := W#16#5521;
   LOG_STORE_DATA[494] := W#16#0;
   LOG_STORE_DATA[495] := W#16#0;
   LOG_STORE_DATA[496] := W#16#400;
   LOG_STORE_DATA[497] := W#16#1310;
   LOG_STORE_DATA[498] := W#16#5511;
   LOG_STORE_DATA[499] := W#16#0;
   LOG_STORE_DATA[500] := W#16#0;
   ORDER_DATA_SWAP[1] := B#16#0;
   ORDER_DATA_SWAP[2] := B#16#0;
   ORDER_DATA_SWAP[3] := B#16#0;
   ORDER_DATA_SWAP[4] := B#16#0;
   ORDER_DATA_SWAP[5] := B#16#0;
   ORDER_DATA_SWAP[6] := B#16#0;
   ORDER_DATA_SWAP[7] := B#16#0;
   ORDER_DATA_SWAP[8] := B#16#0;
   ORDER_DATA_SWAP[9] := B#16#0;
   ORDER_DATA_SWAP[10] := B#16#0;
   ORDER_DATA_SWAP[11] := B#16#0;
   ORDER_DATA_SWAP[12] := B#16#0;
   ORDER_DATA_SWAP[13] := B#16#0;
   ORDER_DATA_SWAP[14] := B#16#0;
   ORDER_DATA_SWAP[15] := B#16#0;
   ORDER_DATA_SWAP[16] := B#16#0;
   TEMP1[1] := B#16#0;
   TEMP1[2] := B#16#0;
   TEMP1[3] := B#16#0;
   TEMP1[4] := B#16#0;
   LINE_PRESENT_SWAP[1] := B#16#0;
   LINE_PRESENT_SWAP[2] := B#16#0;
   LINE_PRESENT_SWAP[3] := B#16#0;
   LINE_PRESENT_SWAP[4] := B#16#0;
   LINE_PRESENT_SWAP[5] := B#16#0;
   LINE_PRESENT_SWAP[6] := B#16#0;
   LINE_PRESENT_SWAP[7] := B#16#0;
   LINE_PRESENT_SWAP[8] := B#16#0;
   LINE_PRESENT_SWAP[9] := B#16#0;
   LINE_PRESENT_SWAP[10] := B#16#0;
   LINE_PRESENT_SWAP[11] := B#16#0;
   LINE_PRESENT_SWAP[12] := B#16#0;
   LINE_PRESENT_SWAP[13] := B#16#0;
   LINE_PRESENT_SWAP[14] := B#16#0;
   LINE_PRESENT_SWAP[15] := B#16#0;
   LINE_PRESENT_SWAP[16] := B#16#0;
END_DATA_BLOCK

DATA_BLOCK DB 162
TITLE =
VERSION : 0.1


  STRUCT
   Compare_VIN_Data1 : WORD ;	//수신 데이터 비교용 임시영역
   Compare_VIN_Data2 : WORD ;	//수신 데이터 비교용 임시영역
   Compare_Body_Data1 : WORD ;	//수신 데이터 비교용 임시영역
   Compare_Body_Data2 : WORD ;	//수신 데이터 비교용 임시영역
   Compare_Body_Data3 : WORD ;	//수신 데이터 비교용 임시영역
   Compare_Body_Data4 : WORD ;	//수신 데이터 비교용 임시영역
   Compare_Body_Data5 : WORD ;	//수신 데이터 비교용 임시영역
   Compare_Body_Data6 : WORD ;	//수신 데이터 비교용 임시영역
   Present_VIN_Data1 : WORD ;	//현재 공정 데이터 저장영역
   Present_VIN_Data2 : WORD ;	//현재 공정 데이터 저장영역
   Present_Body_Data1 : WORD ;	//현재 공정 데이터 저장영역
   Present_Body_Data2 : WORD ;	//현재 공정 데이터 저장영역
   Present_Body_Data3 : WORD ;	//현재 공정 데이터 저장영역
   Present_Body_Data4 : WORD ;	//현재 공정 데이터 저장영역
   Present_Body_Data5 : WORD ;	//현재 공정 데이터 저장영역
   Present_Body_Data6 : WORD ;	//현재 공정 데이터 저장영역
   Communication_Check1 : INT ;	//통신 확인용 1
   Communication_Check2 : INT ;	//통신 확인용 2
   FAC_IF_Data_OldValue : INT ;	//차종 설정 요청 정보 확인용 임시 저장 영역
   unused1 : INT ;
   Read_Date_Time : ARRAY  [1 .. 6 ] OF //PLC 현재 Date&Time Read 후 저장영역
   BYTE ;
   Set_Date_Time : ARRAY  [1 .. 6 ] OF //PLC Date&Time 변경 Data 저장영역
   BYTE ;
   Temporary_Bit : ARRAY  [1 .. 40 ] OF //생산지시용 함수 내부 사용 Bit Memory
   BOOL  := FALSE;
   Temporary_Bit_PLS : ARRAY  [1 .. 40 ] OF //생산지시용 함수 내부 사용 Pulse Bit Memory
   BOOL  := FALSE;
   unused2 : WORD ;
   unused3 : WORD ;
   unused4 : WORD ;
   unused5 : WORD ;
   unused6 : WORD ;
   unused7 : WORD ;
   unused8 : WORD ;
   Temporary : ARRAY  [1 .. 7 ] OF WORD ;
   LOG_LOOP_CNT : INT ;	//LOG저장시 루프 카운터값 저장
   LOG_LOOP_INDEX1 : INT ;	//LOG저장시 MOV포인트 기억용1
   LOG_LOOP_INDEX2 : INT ;	//LOG저장시 MOV포인트 기억용2
   TEMP_INT1 : INT ;
   LOG_STORE_DATA : ARRAY  [1 .. 500 ] OF //로그 저장 영역
   WORD ;
   ORDER_DATA_SWAP : ARRAY  [1 .. 16 ] OF BYTE ;
   TEMP1 : ARRAY  [1 .. 4 ] OF BYTE ;
   LINE_PRESENT_SWAP : ARRAY  [1 .. 16 ] OF BYTE ;
  END_STRUCT ;
BEGIN
   Compare_VIN_Data1 := W#16#4944;
   Compare_VIN_Data2 := W#16#23;
   Compare_Body_Data1 := W#16#A21;
   Compare_Body_Data2 := W#16#1040;
   Compare_Body_Data3 := W#16#4616;
   Compare_Body_Data4 := W#16#0;
   Compare_Body_Data5 := W#16#0;
   Compare_Body_Data6 := W#16#0;
   Present_VIN_Data1 := W#16#23;
   Present_VIN_Data2 := W#16#4943;
   Present_Body_Data1 := W#16#2142;
   Present_Body_Data2 := W#16#8010;
   Present_Body_Data3 := W#16#2A56;
   Present_Body_Data4 := W#16#0;
   Present_Body_Data5 := W#16#0;
   Present_Body_Data6 := W#16#0;
   Communication_Check1 := 0;
   Communication_Check2 := 9;
   FAC_IF_Data_OldValue := 3;
   unused1 := 0;
   Read_Date_Time[1] := B#16#0;
   Read_Date_Time[2] := B#16#0;
   Read_Date_Time[3] := B#16#0;
   Read_Date_Time[4] := B#16#0;
   Read_Date_Time[5] := B#16#0;
   Read_Date_Time[6] := B#16#0;
   Set_Date_Time[1] := B#16#0;
   Set_Date_Time[2] := B#16#0;
   Set_Date_Time[3] := B#16#0;
   Set_Date_Time[4] := B#16#0;
   Set_Date_Time[5] := B#16#0;
   Set_Date_Time[6] := B#16#0;
   Temporary_Bit[1] := FALSE;
   Temporary_Bit[2] := FALSE;
   Temporary_Bit[3] := TRUE;
   Temporary_Bit[4] := FALSE;
   Temporary_Bit[5] := FALSE;
   Temporary_Bit[6] := FALSE;
   Temporary_Bit[7] := FALSE;
   Temporary_Bit[8] := TRUE;
   Temporary_Bit[9] := FALSE;
   Temporary_Bit[10] := FALSE;
   Temporary_Bit[11] := FALSE;
   Temporary_Bit[12] := FALSE;
   Temporary_Bit[13] := FALSE;
   Temporary_Bit[14] := FALSE;
   Temporary_Bit[15] := FALSE;
   Temporary_Bit[16] := FALSE;
   Temporary_Bit[17] := FALSE;
   Temporary_Bit[18] := FALSE;
   Temporary_Bit[19] := FALSE;
   Temporary_Bit[20] := FALSE;
   Temporary_Bit[21] := FALSE;
   Temporary_Bit[22] := FALSE;
   Temporary_Bit[23] := FALSE;
   Temporary_Bit[24] := FALSE;
   Temporary_Bit[25] := FALSE;
   Temporary_Bit[26] := FALSE;
   Temporary_Bit[27] := FALSE;
   Temporary_Bit[28] := FALSE;
   Temporary_Bit[29] := FALSE;
   Temporary_Bit[30] := FALSE;
   Temporary_Bit[31] := FALSE;
   Temporary_Bit[32] := FALSE;
   Temporary_Bit[33] := FALSE;
   Temporary_Bit[34] := FALSE;
   Temporary_Bit[35] := FALSE;
   Temporary_Bit[36] := FALSE;
   Temporary_Bit[37] := FALSE;
   Temporary_Bit[38] := FALSE;
   Temporary_Bit[39] := FALSE;
   Temporary_Bit[40] := FALSE;
   Temporary_Bit_PLS[1] := FALSE;
   Temporary_Bit_PLS[2] := FALSE;
   Temporary_Bit_PLS[3] := TRUE;
   Temporary_Bit_PLS[4] := TRUE;
   Temporary_Bit_PLS[5] := TRUE;
   Temporary_Bit_PLS[6] := FALSE;
   Temporary_Bit_PLS[7] := FALSE;
   Temporary_Bit_PLS[8] := FALSE;
   Temporary_Bit_PLS[9] := FALSE;
   Temporary_Bit_PLS[10] := FALSE;
   Temporary_Bit_PLS[11] := FALSE;
   Temporary_Bit_PLS[12] := FALSE;
   Temporary_Bit_PLS[13] := FALSE;
   Temporary_Bit_PLS[14] := FALSE;
   Temporary_Bit_PLS[15] := FALSE;
   Temporary_Bit_PLS[16] := FALSE;
   Temporary_Bit_PLS[17] := FALSE;
   Temporary_Bit_PLS[18] := FALSE;
   Temporary_Bit_PLS[19] := FALSE;
   Temporary_Bit_PLS[20] := FALSE;
   Temporary_Bit_PLS[21] := FALSE;
   Temporary_Bit_PLS[22] := FALSE;
   Temporary_Bit_PLS[23] := FALSE;
   Temporary_Bit_PLS[24] := FALSE;
   Temporary_Bit_PLS[25] := FALSE;
   Temporary_Bit_PLS[26] := TRUE;
   Temporary_Bit_PLS[27] := FALSE;
   Temporary_Bit_PLS[28] := FALSE;
   Temporary_Bit_PLS[29] := FALSE;
   Temporary_Bit_PLS[30] := FALSE;
   Temporary_Bit_PLS[31] := FALSE;
   Temporary_Bit_PLS[32] := FALSE;
   Temporary_Bit_PLS[33] := FALSE;
   Temporary_Bit_PLS[34] := FALSE;
   Temporary_Bit_PLS[35] := FALSE;
   Temporary_Bit_PLS[36] := FALSE;
   Temporary_Bit_PLS[37] := FALSE;
   Temporary_Bit_PLS[38] := FALSE;
   Temporary_Bit_PLS[39] := FALSE;
   Temporary_Bit_PLS[40] := FALSE;
   unused2 := W#16#0;
   unused3 := W#16#0;
   unused4 := W#16#0;
   unused5 := W#16#0;
   unused6 := W#16#0;
   unused7 := W#16#0;
   unused8 := W#16#0;
   Temporary[1] := W#16#0;
   Temporary[2] := W#16#0;
   Temporary[3] := W#16#0;
   Temporary[4] := W#16#0;
   Temporary[5] := W#16#0;
   Temporary[6] := W#16#0;
   Temporary[7] := W#16#0;
   LOG_LOOP_CNT := 100;
   LOG_LOOP_INDEX1 := 90;
   LOG_LOOP_INDEX2 := 80;
   TEMP_INT1 := 0;
   LOG_STORE_DATA[1] := W#16#400;
   LOG_STORE_DATA[2] := W#16#1715;
   LOG_STORE_DATA[3] := W#16#5943;
   LOG_STORE_DATA[4] := W#16#0;
   LOG_STORE_DATA[5] := W#16#4943;
   LOG_STORE_DATA[6] := W#16#300;
   LOG_STORE_DATA[7] := W#16#1715;
   LOG_STORE_DATA[8] := W#16#5942;
   LOG_STORE_DATA[9] := W#16#B;
   LOG_STORE_DATA[10] := W#16#4943;
   LOG_STORE_DATA[11] := W#16#200;
   LOG_STORE_DATA[12] := W#16#1715;
   LOG_STORE_DATA[13] := W#16#5940;
   LOG_STORE_DATA[14] := W#16#1;
   LOG_STORE_DATA[15] := W#16#4942;
   LOG_STORE_DATA[16] := W#16#500;
   LOG_STORE_DATA[17] := W#16#1715;
   LOG_STORE_DATA[18] := W#16#5939;
   LOG_STORE_DATA[19] := W#16#0;
   LOG_STORE_DATA[20] := W#16#0;
   LOG_STORE_DATA[21] := W#16#400;
   LOG_STORE_DATA[22] := W#16#1715;
   LOG_STORE_DATA[23] := W#16#5825;
   LOG_STORE_DATA[24] := W#16#0;
   LOG_STORE_DATA[25] := W#16#4942;
   LOG_STORE_DATA[26] := W#16#300;
   LOG_STORE_DATA[27] := W#16#1715;
   LOG_STORE_DATA[28] := W#16#5823;
   LOG_STORE_DATA[29] := W#16#B;
   LOG_STORE_DATA[30] := W#16#4942;
   LOG_STORE_DATA[31] := W#16#200;
   LOG_STORE_DATA[32] := W#16#1715;
   LOG_STORE_DATA[33] := W#16#5821;
   LOG_STORE_DATA[34] := W#16#1;
   LOG_STORE_DATA[35] := W#16#4941;
   LOG_STORE_DATA[36] := W#16#500;
   LOG_STORE_DATA[37] := W#16#1715;
   LOG_STORE_DATA[38] := W#16#5820;
   LOG_STORE_DATA[39] := W#16#0;
   LOG_STORE_DATA[40] := W#16#0;
   LOG_STORE_DATA[41] := W#16#400;
   LOG_STORE_DATA[42] := W#16#1715;
   LOG_STORE_DATA[43] := W#16#5653;
   LOG_STORE_DATA[44] := W#16#0;
   LOG_STORE_DATA[45] := W#16#4941;
   LOG_STORE_DATA[46] := W#16#300;
   LOG_STORE_DATA[47] := W#16#1715;
   LOG_STORE_DATA[48] := W#16#5650;
   LOG_STORE_DATA[49] := W#16#B;
   LOG_STORE_DATA[50] := W#16#4941;
   LOG_STORE_DATA[51] := W#16#200;
   LOG_STORE_DATA[52] := W#16#1715;
   LOG_STORE_DATA[53] := W#16#5649;
   LOG_STORE_DATA[54] := W#16#1;
   LOG_STORE_DATA[55] := W#16#4940;
   LOG_STORE_DATA[56] := W#16#500;
   LOG_STORE_DATA[57] := W#16#1715;
   LOG_STORE_DATA[58] := W#16#5648;
   LOG_STORE_DATA[59] := W#16#0;
   LOG_STORE_DATA[60] := W#16#0;
   LOG_STORE_DATA[61] := W#16#400;
   LOG_STORE_DATA[62] := W#16#1715;
   LOG_STORE_DATA[63] := W#16#5535;
   LOG_STORE_DATA[64] := W#16#0;
   LOG_STORE_DATA[65] := W#16#4940;
   LOG_STORE_DATA[66] := W#16#300;
   LOG_STORE_DATA[67] := W#16#1715;
   LOG_STORE_DATA[68] := W#16#5532;
   LOG_STORE_DATA[69] := W#16#B;
   LOG_STORE_DATA[70] := W#16#4940;
   LOG_STORE_DATA[71] := W#16#200;
   LOG_STORE_DATA[72] := W#16#1715;
   LOG_STORE_DATA[73] := W#16#5530;
   LOG_STORE_DATA[74] := W#16#1;
   LOG_STORE_DATA[75] := W#16#4939;
   LOG_STORE_DATA[76] := W#16#500;
   LOG_STORE_DATA[77] := W#16#1715;
   LOG_STORE_DATA[78] := W#16#5530;
   LOG_STORE_DATA[79] := W#16#0;
   LOG_STORE_DATA[80] := W#16#0;
   LOG_STORE_DATA[81] := W#16#400;
   LOG_STORE_DATA[82] := W#16#1715;
   LOG_STORE_DATA[83] := W#16#5350;
   LOG_STORE_DATA[84] := W#16#0;
   LOG_STORE_DATA[85] := W#16#4939;
   LOG_STORE_DATA[86] := W#16#300;
   LOG_STORE_DATA[87] := W#16#1715;
   LOG_STORE_DATA[88] := W#16#5347;
   LOG_STORE_DATA[89] := W#16#B;
   LOG_STORE_DATA[90] := W#16#4939;
   LOG_STORE_DATA[91] := W#16#200;
   LOG_STORE_DATA[92] := W#16#1715;
   LOG_STORE_DATA[93] := W#16#5345;
   LOG_STORE_DATA[94] := W#16#1;
   LOG_STORE_DATA[95] := W#16#4938;
   LOG_STORE_DATA[96] := W#16#500;
   LOG_STORE_DATA[97] := W#16#1715;
   LOG_STORE_DATA[98] := W#16#5344;
   LOG_STORE_DATA[99] := W#16#0;
   LOG_STORE_DATA[100] := W#16#0;
   LOG_STORE_DATA[101] := W#16#400;
   LOG_STORE_DATA[102] := W#16#1715;
   LOG_STORE_DATA[103] := W#16#5231;
   LOG_STORE_DATA[104] := W#16#0;
   LOG_STORE_DATA[105] := W#16#4938;
   LOG_STORE_DATA[106] := W#16#300;
   LOG_STORE_DATA[107] := W#16#1715;
   LOG_STORE_DATA[108] := W#16#5229;
   LOG_STORE_DATA[109] := W#16#B;
   LOG_STORE_DATA[110] := W#16#4938;
   LOG_STORE_DATA[111] := W#16#200;
   LOG_STORE_DATA[112] := W#16#1715;
   LOG_STORE_DATA[113] := W#16#5227;
   LOG_STORE_DATA[114] := W#16#1;
   LOG_STORE_DATA[115] := W#16#4937;
   LOG_STORE_DATA[116] := W#16#500;
   LOG_STORE_DATA[117] := W#16#1715;
   LOG_STORE_DATA[118] := W#16#5226;
   LOG_STORE_DATA[119] := W#16#0;
   LOG_STORE_DATA[120] := W#16#0;
   LOG_STORE_DATA[121] := W#16#400;
   LOG_STORE_DATA[122] := W#16#1715;
   LOG_STORE_DATA[123] := W#16#5114;
   LOG_STORE_DATA[124] := W#16#0;
   LOG_STORE_DATA[125] := W#16#4937;
   LOG_STORE_DATA[126] := W#16#300;
   LOG_STORE_DATA[127] := W#16#1715;
   LOG_STORE_DATA[128] := W#16#5111;
   LOG_STORE_DATA[129] := W#16#B;
   LOG_STORE_DATA[130] := W#16#4937;
   LOG_STORE_DATA[131] := W#16#200;
   LOG_STORE_DATA[132] := W#16#1715;
   LOG_STORE_DATA[133] := W#16#5110;
   LOG_STORE_DATA[134] := W#16#1;
   LOG_STORE_DATA[135] := W#16#4936;
   LOG_STORE_DATA[136] := W#16#500;
   LOG_STORE_DATA[137] := W#16#1715;
   LOG_STORE_DATA[138] := W#16#5109;
   LOG_STORE_DATA[139] := W#16#0;
   LOG_STORE_DATA[140] := W#16#0;
   LOG_STORE_DATA[141] := W#16#400;
   LOG_STORE_DATA[142] := W#16#1715;
   LOG_STORE_DATA[143] := W#16#4951;
   LOG_STORE_DATA[144] := W#16#0;
   LOG_STORE_DATA[145] := W#16#4936;
   LOG_STORE_DATA[146] := W#16#300;
   LOG_STORE_DATA[147] := W#16#1715;
   LOG_STORE_DATA[148] := W#16#4949;
   LOG_STORE_DATA[149] := W#16#B;
   LOG_STORE_DATA[150] := W#16#4936;
   LOG_STORE_DATA[151] := W#16#200;
   LOG_STORE_DATA[152] := W#16#1715;
   LOG_STORE_DATA[153] := W#16#4947;
   LOG_STORE_DATA[154] := W#16#1;
   LOG_STORE_DATA[155] := W#16#4935;
   LOG_STORE_DATA[156] := W#16#500;
   LOG_STORE_DATA[157] := W#16#1715;
   LOG_STORE_DATA[158] := W#16#4946;
   LOG_STORE_DATA[159] := W#16#0;
   LOG_STORE_DATA[160] := W#16#0;
   LOG_STORE_DATA[161] := W#16#400;
   LOG_STORE_DATA[162] := W#16#1715;
   LOG_STORE_DATA[163] := W#16#4831;
   LOG_STORE_DATA[164] := W#16#0;
   LOG_STORE_DATA[165] := W#16#4935;
   LOG_STORE_DATA[166] := W#16#300;
   LOG_STORE_DATA[167] := W#16#1715;
   LOG_STORE_DATA[168] := W#16#4830;
   LOG_STORE_DATA[169] := W#16#B;
   LOG_STORE_DATA[170] := W#16#4935;
   LOG_STORE_DATA[171] := W#16#200;
   LOG_STORE_DATA[172] := W#16#1715;
   LOG_STORE_DATA[173] := W#16#4828;
   LOG_STORE_DATA[174] := W#16#1;
   LOG_STORE_DATA[175] := W#16#4934;
   LOG_STORE_DATA[176] := W#16#500;
   LOG_STORE_DATA[177] := W#16#1715;
   LOG_STORE_DATA[178] := W#16#4827;
   LOG_STORE_DATA[179] := W#16#0;
   LOG_STORE_DATA[180] := W#16#0;
   LOG_STORE_DATA[181] := W#16#400;
   LOG_STORE_DATA[182] := W#16#1715;
   LOG_STORE_DATA[183] := W#16#4342;
   LOG_STORE_DATA[184] := W#16#0;
   LOG_STORE_DATA[185] := W#16#4934;
   LOG_STORE_DATA[186] := W#16#300;
   LOG_STORE_DATA[187] := W#16#1715;
   LOG_STORE_DATA[188] := W#16#4339;
   LOG_STORE_DATA[189] := W#16#B;
   LOG_STORE_DATA[190] := W#16#4934;
   LOG_STORE_DATA[191] := W#16#200;
   LOG_STORE_DATA[192] := W#16#1715;
   LOG_STORE_DATA[193] := W#16#4337;
   LOG_STORE_DATA[194] := W#16#1;
   LOG_STORE_DATA[195] := W#16#4933;
   LOG_STORE_DATA[196] := W#16#500;
   LOG_STORE_DATA[197] := W#16#1715;
   LOG_STORE_DATA[198] := W#16#4336;
   LOG_STORE_DATA[199] := W#16#0;
   LOG_STORE_DATA[200] := W#16#0;
   LOG_STORE_DATA[201] := W#16#400;
   LOG_STORE_DATA[202] := W#16#1715;
   LOG_STORE_DATA[203] := W#16#4223;
   LOG_STORE_DATA[204] := W#16#0;
   LOG_STORE_DATA[205] := W#16#4933;
   LOG_STORE_DATA[206] := W#16#300;
   LOG_STORE_DATA[207] := W#16#1715;
   LOG_STORE_DATA[208] := W#16#4220;
   LOG_STORE_DATA[209] := W#16#B;
   LOG_STORE_DATA[210] := W#16#4933;
   LOG_STORE_DATA[211] := W#16#200;
   LOG_STORE_DATA[212] := W#16#1715;
   LOG_STORE_DATA[213] := W#16#4218;
   LOG_STORE_DATA[214] := W#16#1;
   LOG_STORE_DATA[215] := W#16#4932;
   LOG_STORE_DATA[216] := W#16#500;
   LOG_STORE_DATA[217] := W#16#1715;
   LOG_STORE_DATA[218] := W#16#4217;
   LOG_STORE_DATA[219] := W#16#0;
   LOG_STORE_DATA[220] := W#16#0;
   LOG_STORE_DATA[221] := W#16#400;
   LOG_STORE_DATA[222] := W#16#1715;
   LOG_STORE_DATA[223] := W#16#4056;
   LOG_STORE_DATA[224] := W#16#0;
   LOG_STORE_DATA[225] := W#16#4932;
   LOG_STORE_DATA[226] := W#16#300;
   LOG_STORE_DATA[227] := W#16#1715;
   LOG_STORE_DATA[228] := W#16#4054;
   LOG_STORE_DATA[229] := W#16#B;
   LOG_STORE_DATA[230] := W#16#4932;
   LOG_STORE_DATA[231] := W#16#200;
   LOG_STORE_DATA[232] := W#16#1715;
   LOG_STORE_DATA[233] := W#16#4052;
   LOG_STORE_DATA[234] := W#16#1;
   LOG_STORE_DATA[235] := W#16#4931;
   LOG_STORE_DATA[236] := W#16#500;
   LOG_STORE_DATA[237] := W#16#1715;
   LOG_STORE_DATA[238] := W#16#4051;
   LOG_STORE_DATA[239] := W#16#0;
   LOG_STORE_DATA[240] := W#16#0;
   LOG_STORE_DATA[241] := W#16#400;
   LOG_STORE_DATA[242] := W#16#1715;
   LOG_STORE_DATA[243] := W#16#3912;
   LOG_STORE_DATA[244] := W#16#0;
   LOG_STORE_DATA[245] := W#16#4931;
   LOG_STORE_DATA[246] := W#16#300;
   LOG_STORE_DATA[247] := W#16#1715;
   LOG_STORE_DATA[248] := W#16#3910;
   LOG_STORE_DATA[249] := W#16#B;
   LOG_STORE_DATA[250] := W#16#4931;
   LOG_STORE_DATA[251] := W#16#200;
   LOG_STORE_DATA[252] := W#16#1715;
   LOG_STORE_DATA[253] := W#16#3908;
   LOG_STORE_DATA[254] := W#16#1;
   LOG_STORE_DATA[255] := W#16#4930;
   LOG_STORE_DATA[256] := W#16#500;
   LOG_STORE_DATA[257] := W#16#1715;
   LOG_STORE_DATA[258] := W#16#3907;
   LOG_STORE_DATA[259] := W#16#0;
   LOG_STORE_DATA[260] := W#16#0;
   LOG_STORE_DATA[261] := W#16#400;
   LOG_STORE_DATA[262] := W#16#1715;
   LOG_STORE_DATA[263] := W#16#3739;
   LOG_STORE_DATA[264] := W#16#0;
   LOG_STORE_DATA[265] := W#16#4930;
   LOG_STORE_DATA[266] := W#16#300;
   LOG_STORE_DATA[267] := W#16#1715;
   LOG_STORE_DATA[268] := W#16#3736;
   LOG_STORE_DATA[269] := W#16#B;
   LOG_STORE_DATA[270] := W#16#4930;
   LOG_STORE_DATA[271] := W#16#200;
   LOG_STORE_DATA[272] := W#16#1715;
   LOG_STORE_DATA[273] := W#16#3734;
   LOG_STORE_DATA[274] := W#16#1;
   LOG_STORE_DATA[275] := W#16#4929;
   LOG_STORE_DATA[276] := W#16#500;
   LOG_STORE_DATA[277] := W#16#1715;
   LOG_STORE_DATA[278] := W#16#3733;
   LOG_STORE_DATA[279] := W#16#0;
   LOG_STORE_DATA[280] := W#16#0;
   LOG_STORE_DATA[281] := W#16#400;
   LOG_STORE_DATA[282] := W#16#1715;
   LOG_STORE_DATA[283] := W#16#3618;
   LOG_STORE_DATA[284] := W#16#0;
   LOG_STORE_DATA[285] := W#16#4929;
   LOG_STORE_DATA[286] := W#16#300;
   LOG_STORE_DATA[287] := W#16#1715;
   LOG_STORE_DATA[288] := W#16#3616;
   LOG_STORE_DATA[289] := W#16#B;
   LOG_STORE_DATA[290] := W#16#4929;
   LOG_STORE_DATA[291] := W#16#200;
   LOG_STORE_DATA[292] := W#16#1715;
   LOG_STORE_DATA[293] := W#16#3614;
   LOG_STORE_DATA[294] := W#16#1;
   LOG_STORE_DATA[295] := W#16#4928;
   LOG_STORE_DATA[296] := W#16#500;
   LOG_STORE_DATA[297] := W#16#1715;
   LOG_STORE_DATA[298] := W#16#3613;
   LOG_STORE_DATA[299] := W#16#0;
   LOG_STORE_DATA[300] := W#16#0;
   LOG_STORE_DATA[301] := W#16#400;
   LOG_STORE_DATA[302] := W#16#1715;
   LOG_STORE_DATA[303] := W#16#3409;
   LOG_STORE_DATA[304] := W#16#0;
   LOG_STORE_DATA[305] := W#16#4928;
   LOG_STORE_DATA[306] := W#16#300;
   LOG_STORE_DATA[307] := W#16#1715;
   LOG_STORE_DATA[308] := W#16#3406;
   LOG_STORE_DATA[309] := W#16#B;
   LOG_STORE_DATA[310] := W#16#4928;
   LOG_STORE_DATA[311] := W#16#200;
   LOG_STORE_DATA[312] := W#16#1715;
   LOG_STORE_DATA[313] := W#16#3405;
   LOG_STORE_DATA[314] := W#16#1;
   LOG_STORE_DATA[315] := W#16#4927;
   LOG_STORE_DATA[316] := W#16#500;
   LOG_STORE_DATA[317] := W#16#1715;
   LOG_STORE_DATA[318] := W#16#3403;
   LOG_STORE_DATA[319] := W#16#0;
   LOG_STORE_DATA[320] := W#16#0;
   LOG_STORE_DATA[321] := W#16#400;
   LOG_STORE_DATA[322] := W#16#1715;
   LOG_STORE_DATA[323] := W#16#3249;
   LOG_STORE_DATA[324] := W#16#0;
   LOG_STORE_DATA[325] := W#16#4927;
   LOG_STORE_DATA[326] := W#16#300;
   LOG_STORE_DATA[327] := W#16#1715;
   LOG_STORE_DATA[328] := W#16#3246;
   LOG_STORE_DATA[329] := W#16#B;
   LOG_STORE_DATA[330] := W#16#4927;
   LOG_STORE_DATA[331] := W#16#200;
   LOG_STORE_DATA[332] := W#16#1715;
   LOG_STORE_DATA[333] := W#16#3244;
   LOG_STORE_DATA[334] := W#16#1;
   LOG_STORE_DATA[335] := W#16#4926;
   LOG_STORE_DATA[336] := W#16#500;
   LOG_STORE_DATA[337] := W#16#1715;
   LOG_STORE_DATA[338] := W#16#3243;
   LOG_STORE_DATA[339] := W#16#0;
   LOG_STORE_DATA[340] := W#16#0;
   LOG_STORE_DATA[341] := W#16#400;
   LOG_STORE_DATA[342] := W#16#1715;
   LOG_STORE_DATA[343] := W#16#3021;
   LOG_STORE_DATA[344] := W#16#0;
   LOG_STORE_DATA[345] := W#16#4926;
   LOG_STORE_DATA[346] := W#16#300;
   LOG_STORE_DATA[347] := W#16#1715;
   LOG_STORE_DATA[348] := W#16#3019;
   LOG_STORE_DATA[349] := W#16#B;
   LOG_STORE_DATA[350] := W#16#4926;
   LOG_STORE_DATA[351] := W#16#200;
   LOG_STORE_DATA[352] := W#16#1715;
   LOG_STORE_DATA[353] := W#16#3018;
   LOG_STORE_DATA[354] := W#16#1;
   LOG_STORE_DATA[355] := W#16#4925;
   LOG_STORE_DATA[356] := W#16#500;
   LOG_STORE_DATA[357] := W#16#1715;
   LOG_STORE_DATA[358] := W#16#3017;
   LOG_STORE_DATA[359] := W#16#0;
   LOG_STORE_DATA[360] := W#16#0;
   LOG_STORE_DATA[361] := W#16#400;
   LOG_STORE_DATA[362] := W#16#1715;
   LOG_STORE_DATA[363] := W#16#2903;
   LOG_STORE_DATA[364] := W#16#0;
   LOG_STORE_DATA[365] := W#16#4925;
   LOG_STORE_DATA[366] := W#16#300;
   LOG_STORE_DATA[367] := W#16#1715;
   LOG_STORE_DATA[368] := W#16#2900;
   LOG_STORE_DATA[369] := W#16#B;
   LOG_STORE_DATA[370] := W#16#4925;
   LOG_STORE_DATA[371] := W#16#200;
   LOG_STORE_DATA[372] := W#16#1715;
   LOG_STORE_DATA[373] := W#16#2858;
   LOG_STORE_DATA[374] := W#16#1;
   LOG_STORE_DATA[375] := W#16#4924;
   LOG_STORE_DATA[376] := W#16#500;
   LOG_STORE_DATA[377] := W#16#1715;
   LOG_STORE_DATA[378] := W#16#2857;
   LOG_STORE_DATA[379] := W#16#0;
   LOG_STORE_DATA[380] := W#16#0;
   LOG_STORE_DATA[381] := W#16#400;
   LOG_STORE_DATA[382] := W#16#1715;
   LOG_STORE_DATA[383] := W#16#2736;
   LOG_STORE_DATA[384] := W#16#0;
   LOG_STORE_DATA[385] := W#16#4924;
   LOG_STORE_DATA[386] := W#16#300;
   LOG_STORE_DATA[387] := W#16#1715;
   LOG_STORE_DATA[388] := W#16#2735;
   LOG_STORE_DATA[389] := W#16#B;
   LOG_STORE_DATA[390] := W#16#4924;
   LOG_STORE_DATA[391] := W#16#200;
   LOG_STORE_DATA[392] := W#16#1715;
   LOG_STORE_DATA[393] := W#16#2733;
   LOG_STORE_DATA[394] := W#16#1;
   LOG_STORE_DATA[395] := W#16#4923;
   LOG_STORE_DATA[396] := W#16#500;
   LOG_STORE_DATA[397] := W#16#1715;
   LOG_STORE_DATA[398] := W#16#2732;
   LOG_STORE_DATA[399] := W#16#0;
   LOG_STORE_DATA[400] := W#16#0;
   LOG_STORE_DATA[401] := W#16#400;
   LOG_STORE_DATA[402] := W#16#1715;
   LOG_STORE_DATA[403] := W#16#2553;
   LOG_STORE_DATA[404] := W#16#0;
   LOG_STORE_DATA[405] := W#16#4923;
   LOG_STORE_DATA[406] := W#16#300;
   LOG_STORE_DATA[407] := W#16#1715;
   LOG_STORE_DATA[408] := W#16#2550;
   LOG_STORE_DATA[409] := W#16#B;
   LOG_STORE_DATA[410] := W#16#4923;
   LOG_STORE_DATA[411] := W#16#200;
   LOG_STORE_DATA[412] := W#16#1715;
   LOG_STORE_DATA[413] := W#16#2548;
   LOG_STORE_DATA[414] := W#16#1;
   LOG_STORE_DATA[415] := W#16#4922;
   LOG_STORE_DATA[416] := W#16#500;
   LOG_STORE_DATA[417] := W#16#1715;
   LOG_STORE_DATA[418] := W#16#2547;
   LOG_STORE_DATA[419] := W#16#0;
   LOG_STORE_DATA[420] := W#16#0;
   LOG_STORE_DATA[421] := W#16#400;
   LOG_STORE_DATA[422] := W#16#1715;
   LOG_STORE_DATA[423] := W#16#2431;
   LOG_STORE_DATA[424] := W#16#0;
   LOG_STORE_DATA[425] := W#16#4922;
   LOG_STORE_DATA[426] := W#16#300;
   LOG_STORE_DATA[427] := W#16#1715;
   LOG_STORE_DATA[428] := W#16#2428;
   LOG_STORE_DATA[429] := W#16#B;
   LOG_STORE_DATA[430] := W#16#4922;
   LOG_STORE_DATA[431] := W#16#200;
   LOG_STORE_DATA[432] := W#16#1715;
   LOG_STORE_DATA[433] := W#16#2426;
   LOG_STORE_DATA[434] := W#16#1;
   LOG_STORE_DATA[435] := W#16#4921;
   LOG_STORE_DATA[436] := W#16#500;
   LOG_STORE_DATA[437] := W#16#1715;
   LOG_STORE_DATA[438] := W#16#2425;
   LOG_STORE_DATA[439] := W#16#0;
   LOG_STORE_DATA[440] := W#16#0;
   LOG_STORE_DATA[441] := W#16#400;
   LOG_STORE_DATA[442] := W#16#1715;
   LOG_STORE_DATA[443] := W#16#2313;
   LOG_STORE_DATA[444] := W#16#0;
   LOG_STORE_DATA[445] := W#16#4921;
   LOG_STORE_DATA[446] := W#16#300;
   LOG_STORE_DATA[447] := W#16#1715;
   LOG_STORE_DATA[448] := W#16#2310;
   LOG_STORE_DATA[449] := W#16#B;
   LOG_STORE_DATA[450] := W#16#4921;
   LOG_STORE_DATA[451] := W#16#200;
   LOG_STORE_DATA[452] := W#16#1715;
   LOG_STORE_DATA[453] := W#16#2308;
   LOG_STORE_DATA[454] := W#16#1;
   LOG_STORE_DATA[455] := W#16#4920;
   LOG_STORE_DATA[456] := W#16#500;
   LOG_STORE_DATA[457] := W#16#1715;
   LOG_STORE_DATA[458] := W#16#2307;
   LOG_STORE_DATA[459] := W#16#0;
   LOG_STORE_DATA[460] := W#16#0;
   LOG_STORE_DATA[461] := W#16#400;
   LOG_STORE_DATA[462] := W#16#1715;
   LOG_STORE_DATA[463] := W#16#2135;
   LOG_STORE_DATA[464] := W#16#0;
   LOG_STORE_DATA[465] := W#16#4920;
   LOG_STORE_DATA[466] := W#16#300;
   LOG_STORE_DATA[467] := W#16#1715;
   LOG_STORE_DATA[468] := W#16#2133;
   LOG_STORE_DATA[469] := W#16#B;
   LOG_STORE_DATA[470] := W#16#4920;
   LOG_STORE_DATA[471] := W#16#200;
   LOG_STORE_DATA[472] := W#16#1715;
   LOG_STORE_DATA[473] := W#16#2131;
   LOG_STORE_DATA[474] := W#16#1;
   LOG_STORE_DATA[475] := W#16#4919;
   LOG_STORE_DATA[476] := W#16#500;
   LOG_STORE_DATA[477] := W#16#1715;
   LOG_STORE_DATA[478] := W#16#2130;
   LOG_STORE_DATA[479] := W#16#0;
   LOG_STORE_DATA[480] := W#16#0;
   LOG_STORE_DATA[481] := W#16#400;
   LOG_STORE_DATA[482] := W#16#1715;
   LOG_STORE_DATA[483] := W#16#2017;
   LOG_STORE_DATA[484] := W#16#0;
   LOG_STORE_DATA[485] := W#16#4919;
   LOG_STORE_DATA[486] := W#16#300;
   LOG_STORE_DATA[487] := W#16#1715;
   LOG_STORE_DATA[488] := W#16#2015;
   LOG_STORE_DATA[489] := W#16#B;
   LOG_STORE_DATA[490] := W#16#4919;
   LOG_STORE_DATA[491] := W#16#200;
   LOG_STORE_DATA[492] := W#16#1715;
   LOG_STORE_DATA[493] := W#16#2013;
   LOG_STORE_DATA[494] := W#16#1;
   LOG_STORE_DATA[495] := W#16#4918;
   LOG_STORE_DATA[496] := W#16#500;
   LOG_STORE_DATA[497] := W#16#1715;
   LOG_STORE_DATA[498] := W#16#2012;
   LOG_STORE_DATA[499] := W#16#0;
   LOG_STORE_DATA[500] := W#16#0;
   ORDER_DATA_SWAP[1] := B#16#0;
   ORDER_DATA_SWAP[2] := B#16#23;
   ORDER_DATA_SWAP[3] := B#16#49;
   ORDER_DATA_SWAP[4] := B#16#43;
   ORDER_DATA_SWAP[5] := B#16#21;
   ORDER_DATA_SWAP[6] := B#16#42;
   ORDER_DATA_SWAP[7] := B#16#80;
   ORDER_DATA_SWAP[8] := B#16#10;
   ORDER_DATA_SWAP[9] := B#16#2A;
   ORDER_DATA_SWAP[10] := B#16#56;
   ORDER_DATA_SWAP[11] := B#16#0;
   ORDER_DATA_SWAP[12] := B#16#0;
   ORDER_DATA_SWAP[13] := B#16#0;
   ORDER_DATA_SWAP[14] := B#16#0;
   ORDER_DATA_SWAP[15] := B#16#0;
   ORDER_DATA_SWAP[16] := B#16#0;
   TEMP1[1] := B#16#0;
   TEMP1[2] := B#16#0;
   TEMP1[3] := B#16#0;
   TEMP1[4] := B#16#0;
   LINE_PRESENT_SWAP[1] := B#16#49;
   LINE_PRESENT_SWAP[2] := B#16#43;
   LINE_PRESENT_SWAP[3] := B#16#0;
   LINE_PRESENT_SWAP[4] := B#16#23;
   LINE_PRESENT_SWAP[5] := B#16#42;
   LINE_PRESENT_SWAP[6] := B#16#21;
   LINE_PRESENT_SWAP[7] := B#16#10;
   LINE_PRESENT_SWAP[8] := B#16#80;
   LINE_PRESENT_SWAP[9] := B#16#56;
   LINE_PRESENT_SWAP[10] := B#16#2A;
   LINE_PRESENT_SWAP[11] := B#16#0;
   LINE_PRESENT_SWAP[12] := B#16#0;
   LINE_PRESENT_SWAP[13] := B#16#0;
   LINE_PRESENT_SWAP[14] := B#16#0;
   LINE_PRESENT_SWAP[15] := B#16#0;
   LINE_PRESENT_SWAP[16] := B#16#0;
END_DATA_BLOCK

DATA_BLOCK DB 163
TITLE =
VERSION : 0.1


